	{attribute 'TcIecLibraryType'}
	{attribute 'external_name' := 'F_VN_SeparableCustomFilter_GUID_F80F76A2_7DC4_B08F_5EFC_37C20BB33E5D'}
	(* Apply a separable custom filter to the image. *)
	FUNCTION F_VN_SeparableCustomFilter : HRESULT
	VAR_INPUT
		ipSrcImage	:	ITcVnImage;	(* Source image *)
		ipDestImage	:	REFERENCE TO ITcVnImage;	(* Destination image (An appropriate destination image will be created if required.) *)
		eDestDepth	:	ETcVnElementType;	(* Destination image depth *)
	END_VAR
	VAR_IN_OUT
		stKernelX	:	TcVnMatrix;	(* 1D custom row-filter kernel with values of type REAL or LREAL *)
		stKernelY	:	TcVnMatrix;	(* 1D custom column-filter kernel with values of type REAL or LREAL *)
	END_VAR
	VAR_INPUT
		hrPrev	:	HRESULT;	(* HRESULT indicating the result of previous operations (If SUCCEEDED(hrPrev) equals false, no operation is executed.) *)
	END_VAR

END_FUNCTION

// Functions/Image Filtering/F_VN_SeparableCustomFilterExp

	{attribute 'TcIecLibraryType'}
	{attribute 'external_name' := 'F_VN_SeparableCustomFilterExp_GUID_57DB5838_7C15_B21B_75E4_43EDAA86B2A3'}
	(* Apply a separable custom filter to the image. (expert function) *)
	FUNCTION F_VN_SeparableCustomFilterExp : HRESULT
	VAR_INPUT
		ipSrcImage	:	ITcVnImage;	(* Source image *)
		ipDestImage	:	REFERENCE TO ITcVnImage;	(* Destination image (An appropriate destination image will be created if required.) *)
		eDestDepth	:	ETcVnElementType;	(* Destination image depth *)
	END_VAR
	VAR_IN_OUT
		stKernelX	:	TcVnMatrix;	(* 1D custom row-filter kernel with values of type REAL or LREAL *)
		stKernelY	:	TcVnMatrix;	(* 1D custom column-filter kernel with values of type REAL or LREAL *)
		aAnchor	:	TcVnPoint;	(* Anchor point of the kernel *)
	END_VAR
	VAR_INPUT
		fDelta	:	LREAL;	(* Value added to each pixel after filtering *)
		eBorderType	:	ETcVnBorderInterpolationMethod;	(* Image border handling *)
		hrPrev	:	HRESULT;	(* HRESULT indicating the result of previous operations (If SUCCEEDED(hrPrev) equals false, no operation is executed.) *)
	END_VAR

END_FUNCTION

// Functions/Image Filtering/F_VN_SobelFilter

	{attribute 'TcIecLibraryType'}
	{attribute 'external_name' := 'F_VN_SobelFilter_GUID_E336C8FF_820D_B834_7CC9_D468EFC4DB68'}
	(* Calculates the first, second, or mixed image derivatives using an extended Sobel filter. *)
	FUNCTION F_VN_SobelFilter : HRESULT
	VAR_INPUT
		ipSrcImage	:	ITcVnImage;	(* Source image *)
		ipDestImage	:	REFERENCE TO ITcVnImage;	(* Destination image (An appropriate destination image will be created if required.) *)
		eDestDepth	:	ETcVnElementType;	(* Destination image depth *)
		nXOrder	:	UDINT;	(* Order of the x-derivative (0, 1, 2) *)
		nYOrder	:	UDINT;	(* Order of the y-derivative (0, 1, 2) *)
		hrPrev	:	HRESULT;	(* HRESULT indicating the result of previous operations (If SUCCEEDED(hrPrev) equals false, no operation is executed.) *)
	END_VAR

END_FUNCTION

// Functions/Image Filtering/F_VN_SobelFilterExp

	{attribute 'TcIecLibraryType'}
	{attribute 'external_name' := 'F_VN_SobelFilterExp_GUID_605EE3A3_E974_B5AB_57D7_E3CF0E6E55DF'}
	(* Calculates the first, second, third, or mixed image derivatives using an extended Sobel filter. (expert function) *)
	FUNCTION F_VN_SobelFilterExp : HRESULT
	VAR_INPUT
		ipSrcImage	:	ITcVnImage;	(* Source image *)
		ipDestImage	:	REFERENCE TO ITcVnImage;	(* Destination image (An appropriate destination image will be created if required.) *)
		eDestDepth	:	ETcVnElementType;	(* Destination image depth *)
		nXOrder	:	UDINT;	(* Order of the x-derivative (must be < nKernelSize) *)
		nYOrder	:	UDINT;	(* Order of the y-derivative (must be < nKernelSize) *)
		nKernelSize	:	UDINT;	(* Size of the extended Sobel kernel (3, 5, 7, ..., 31) *)
		fScale	:	LREAL;	(* Scale factor for the computed derivative values *)
		fDelta	:	LREAL;	(* Delta value that is added to the results prior to storing them in dest *)
		eBorderType	:	ETcVnBorderInterpolationMethod;	(* Image border handling *)
		hrPrev	:	HRESULT;	(* HRESULT indicating the result of previous operations (If SUCCEEDED(hrPrev) equals false, no operation is executed.) *)
	END_VAR

END_FUNCTION

// Functions/Image Filtering/F_VN_VarianceFilter

	{attribute 'TcIecLibraryType'}
	{attribute 'external_name' := 'F_VN_VarianceFilter_GUID_E9DC81B8_162C_BF12_6F44_85E88F794313'}
	(* Calculates the local variance of an image. *)
	FUNCTION F_VN_VarianceFilter : HRESULT
	VAR_INPUT
		ipSrcImage	:	ITcVnImage;	(* Source image. Only TCVN_ET_USINT Type is supported.  *)
		ipDestImage	:	REFERENCE TO ITcVnImage;	(* Destination image of type TCVN_ET_UINT (An appropriate destination image will be created if required.) *)
		nKernelSize	:	UDINT;	(* Size of the kernel *)
		hrPrev	:	HRESULT;	(* HRESULT indicating the result of previous operations (If SUCCEEDED(hrPrev) equals false, no operation is executed.) *)
	END_VAR

END_FUNCTION

// Functions/Image Filtering/F_VN_VarianceFilterExp

	{attribute 'TcIecLibraryType'}
	{attribute 'external_name' := 'F_VN_VarianceFilterExp_GUID_A3D4813E_C46F_B737_4BEF_710F1779B2AC'}
	(* Calculates the local variance of an image. (expert function) *)
	FUNCTION F_VN_VarianceFilterExp : HRESULT
	VAR_INPUT
		ipSrcImage	:	ITcVnImage;	(* Source image. Only TCVN_ET_USINT Type is supported. *)
		ipDestImage	:	REFERENCE TO ITcVnImage;	(* Destination image of type TCVN_ET_UINT (An appropriate destination image will be created if required.) *)
		nKernelSize	:	UDINT;	(* Size of the kernel *)
		fScale	:	LREAL;	(* Scale factor for the computed variance values *)
		eBorderType	:	ETcVnBorderInterpolationMethod;	(* Image border handling *)
		hrPrev	:	HRESULT;	(* HRESULT indicating the result of previous operations (If SUCCEEDED(hrPrev) equals false, no operation is executed.) *)
	END_VAR

END_FUNCTION

// Functions/Miscellaneous/F_VN_CheckFunctionInitialization

	{attribute 'TcIecLibraryType'}
	{attribute 'external_name' := 'F_VN_CheckFunctionInitialization_GUID_C79D8AB7_DFA6_B5A0_6949_373851CC2509'}
	(* Check if a function is initialized with the specified options. *)
	FUNCTION F_VN_CheckFunctionInitialization : HRESULT
	VAR_INPUT
		eFunction	:	ETcVnInitializableFunction;	(* Initializable function *)
		nOptions	:	ULINT;	(* Initialization options for the function *)
		hrPrev	:	HRESULT;	(* HRESULT indicating the result of previous operations (If SUCCEEDED(hrPrev) equals false, no operation is executed.) *)
	END_VAR

END_FUNCTION

// Functions/Miscellaneous/F_VN_ClipLineToBoundary

	{attribute 'TcIecLibraryType'}
	{attribute 'external_name' := 'F_VN_ClipLineToBoundary_GUID_5F9D10BB_2D68_B024_7AB3_03DA1DD51379'}
	(* Clips a line to a rectangular boundary. *)
	FUNCTION F_VN_ClipLineToBoundary : HRESULT
	VAR_IN_OUT
		aLine	:	TcVnVector4_LREAL;	(* The first and second element describe the x and y component of the direction vector. The third and fourth element describe the x and y component of the position vector. *)
	END_VAR
	VAR_INPUT
		nX1	:	DINT;	(* x of top left rectangle point *)
		nY1	:	DINT;	(* y of top left rectangle point *)
		nX2	:	DINT;	(* x of bottom right rectangle point *)
		nY2	:	DINT;	(* Y of bottom right rectangle point *)
	END_VAR
	VAR_IN_OUT
		aStartPoint	:	TcVnPoint2_REAL;	(* Returns the clipped starting point of the line. *)
		aEndPoint	:	TcVnPoint2_REAL;	(* Returns the clipped end point of the line. *)
	END_VAR
	VAR_INPUT
		hrPrev	:	HRESULT;	(* HRESULT indicating the result of previous operations (If SUCCEEDED(hrPrev) equals false, no operation is executed.) *)
	END_VAR

END_FUNCTION

// Functions/Miscellaneous/F_VN_ClipLineToBoundary_ITcVnImage

	{attribute 'TcIecLibraryType'}
	{attribute 'external_name' := 'F_VN_ClipLineToBoundary_ITcVnImage_GUID_E4D5824B_2FCE_B7A7_6026_B15E63E74A8F'}
	(* Clips a line to the boundary of an image. *)
	FUNCTION F_VN_ClipLineToBoundary_ITcVnImage : HRESULT
	VAR_IN_OUT
		aLine	:	TcVnVector4_LREAL;	(* The first and second element describe the x and y component of the direction vector. The third and fourth element describe the x and y component of the position vector. *)
	END_VAR
	VAR_INPUT
		ipImage	:	ITcVnImage;	(* Image, from which to derive the boundary *)
	END_VAR
	VAR_IN_OUT
		aStartPoint	:	TcVnPoint2_REAL;	(* Returns the clipped starting point of the line. *)
		aEndPoint	:	TcVnPoint2_REAL;	(* Returns the clipped end point of the line. *)
	END_VAR
	VAR_INPUT
		hrPrev	:	HRESULT;	(* HRESULT indicating the result of previous operations (If SUCCEEDED(hrPrev) equals false, no operation is executed.) *)
	END_VAR

END_FUNCTION

// Functions/Miscellaneous/F_VN_ClipLineToBoundary_TcVnRectangle_DINT

	{attribute 'TcIecLibraryType'}
	{attribute 'external_name' := 'F_VN_ClipLineToBoundary_TcVnRectangle_DINT_GUID_87153F32_B3BD_B6D4_74D3_8036D7A03AEC'}
	(* Clips a line to a rectangular boundary. *)
	FUNCTION F_VN_ClipLineToBoundary_TcVnRectangle_DINT : HRESULT
	VAR_IN_OUT
		aLine	:	TcVnVector4_LREAL;	(* The first and second element describe the x and y component of the direction vector. The third and fourth element describe the x and y component of the position vector. *)
		stRectangle	:	TcVnRectangle_DINT;	(* Rectangular boundary *)
		aStartPoint	:	TcVnPoint2_REAL;	(* Returns the clipped starting point of the line. *)
		aEndPoint	:	TcVnPoint2_REAL;	(* Returns the clipped end point of the line. *)
	END_VAR
	VAR_INPUT
		hrPrev	:	HRESULT;	(* HRESULT indicating the result of previous operations (If SUCCEEDED(hrPrev) equals false, no operation is executed.) *)
	END_VAR

END_FUNCTION

// Functions/Miscellaneous/F_VN_ConvertITcUnknownToITcVnBitmapExport

	{attribute 'TcIecLibraryType'}
	{attribute 'external_name' := 'F_VN_ConvertITcUnknownToITcVnBitmapExport_GUID_2EB3F845_B1C8_B651_6556_4CA6475660E3'}
	(* Convert an ITcUnknown interface pointer to an ITcVnBitmapExport interface pointer. The destination pointer will be released (if existing) and set to the source pointer. The source pointer will be set to 0. *)
	FUNCTION F_VN_ConvertITcUnknownToITcVnBitmapExport : HRESULT
	VAR_INPUT
		ipSrc	:	REFERENCE TO ITcUnknown;	(* Source pointer *)
		ipDest	:	REFERENCE TO ITcVnBitmapExport;	(* Destination pointer *)
		hrPrev	:	HRESULT;	(* HRESULT indicating the result of previous operations (If SUCCEEDED(hrPrev) equals false, no operation is executed.) *)
	END_VAR

END_FUNCTION

// Functions/Miscellaneous/F_VN_ConvertITcUnknownToITcVnContainer

	{attribute 'TcIecLibraryType'}
	{attribute 'external_name' := 'F_VN_ConvertITcUnknownToITcVnContainer_GUID_138FA1B4_D6BC_B0DA_5E49_0E92D1E26E82'}
	(* Convert an ITcUnknown interface pointer to an ITcVnContainer interface pointer. The destination pointer will be released (if existing) and set to the source pointer. The source pointer will be set to 0. *)
	FUNCTION F_VN_ConvertITcUnknownToITcVnContainer : HRESULT
	VAR_INPUT
		ipSrc	:	REFERENCE TO ITcUnknown;	(* Source pointer *)
		ipDest	:	REFERENCE TO ITcVnContainer;	(* Destination pointer *)
		hrPrev	:	HRESULT;	(* HRESULT indicating the result of previous operations (If SUCCEEDED(hrPrev) equals false, no operation is executed.) *)
	END_VAR

END_FUNCTION

// Functions/Miscellaneous/F_VN_ConvertITcUnknownToITcVnImage

	{attribute 'TcIecLibraryType'}
	{attribute 'external_name' := 'F_VN_ConvertITcUnknownToITcVnImage_GUID_1C77EE9B_F836_B880_71E3_3B6B684F7DE7'}
	(* Convert an ITcUnknown interface pointer to an ITcVnImage interface pointer. The destination pointer will be released (if existing) and set to the source pointer. The source pointer will be set to 0. *)
	FUNCTION F_VN_ConvertITcUnknownToITcVnImage : HRESULT
	VAR_INPUT
		ipSrc	:	REFERENCE TO ITcUnknown;	(* Source pointer *)
		ipDest	:	REFERENCE TO ITcVnImage;	(* Destination pointer *)
		hrPrev	:	HRESULT;	(* HRESULT indicating the result of previous operations (If SUCCEEDED(hrPrev) equals false, no operation is executed.) *)
	END_VAR

END_FUNCTION

// Functions/Miscellaneous/F_VN_ConvertITcUnknownToITcVnMlModel

	{attribute 'TcIecLibraryType'}
	{attribute 'external_name' := 'F_VN_ConvertITcUnknownToITcVnMlModel_GUID_00F937E1_B5BF_BE31_604E_B90F05C045F2'}
	(* Convert an ITcUnknown interface pointer to an ITcVnMlModel interface pointer. The destination pointer will be released (if existing) and set to the source pointer. The source pointer will be set to 0. *)
	FUNCTION F_VN_ConvertITcUnknownToITcVnMlModel : HRESULT
	VAR_INPUT
		ipSrc	:	REFERENCE TO ITcUnknown;	(* Source pointer *)
		ipDest	:	REFERENCE TO ITcVnMlModel;	(* Destination pointer *)
		hrPrev	:	HRESULT;	(* HRESULT indicating the result of previous operations (If SUCCEEDED(hrPrev) equals false, no operation is executed.) *)
	END_VAR

END_FUNCTION

// Functions/Miscellaneous/F_VN_DeinitializeFunction

	{attribute 'TcIecLibraryType'}
	{attribute 'external_name' := 'F_VN_DeinitializeFunction_GUID_3AEC9F0B_9689_B047_59F3_4962202BFD13'}
	(* Deinitialize the specified options for the function. *)
	FUNCTION F_VN_DeinitializeFunction : HRESULT
	VAR_INPUT
		eFunction	:	ETcVnInitializableFunction;	(* Initializable function *)
		nOptions	:	ULINT;	(* Initialization options for the function *)
		hrPrev	:	HRESULT;	(* HRESULT indicating the result of previous operations (If SUCCEEDED(hrPrev) equals false, no operation is executed.) *)
	END_VAR

END_FUNCTION

// Functions/Miscellaneous/F_VN_GetTimestamp

	{attribute 'TcIecLibraryType'}
	{attribute 'external_name' := 'F_VN_GetTimestamp_GUID_C6774F0F_1FD8_B43F_4215_84A6E64C27D7'}
	(* Get the timestamp (actual DC time) from the last change of an object (e.g. ITcVnImage or ITcVnContainer) *)
	FUNCTION F_VN_GetTimestamp : HRESULT
	VAR_INPUT
		ipUnknown	:	ITcUnknown;	(* An object implementing ITcUnknown and ITcVnTimestamp (e.g. ITcVnImage or ITcVnContainer) *)
	END_VAR
	VAR_IN_OUT
		nTimestamp	:	LINT;	(* Returns the timestamp *)
	END_VAR
	VAR_INPUT
		hrPrev	:	HRESULT;	(* HRESULT indicating the result of previous operations (If SUCCEEDED(hrPrev) equals false, no operation is executed.) *)
	END_VAR

END_FUNCTION

// Functions/Miscellaneous/F_VN_HuMomentInvariants

	{attribute 'TcIecLibraryType'}
	{attribute 'external_name' := 'F_VN_HuMomentInvariants_GUID_BC907807_859C_B8CF_4281_4253B572D82F'}
	(* Computes the Hu moment invariants. *)
	FUNCTION F_VN_HuMomentInvariants : HRESULT
	VAR_IN_OUT
		stMoments	:	TcVnMoments;	(* Moments from which to compute the Hu invariants *)
		aHuInvariants	:	TcVnArray7_LREAL;	(* Returns the Hu moment invariants *)
	END_VAR
	VAR_INPUT
		hrPrev	:	HRESULT;	(* HRESULT indicating the result of previous operations (If SUCCEEDED(hrPrev) equals false, no operation is executed.) *)
	END_VAR

END_FUNCTION

// Functions/Miscellaneous/F_VN_InitMatrixStruct

	{attribute 'TcIecLibraryType'}
	{attribute 'external_name' := 'F_VN_InitMatrixStruct_GUID_8788B85B_B119_B982_4540_76E6A59BE885'}
	(* Initialize a struct of the type TcVnMatrix extending a buffer with metainformation so that it can be used as a matrix. *)
	FUNCTION F_VN_InitMatrixStruct : HRESULT
	VAR_INPUT
		pSrcBuffer	:	PVOID;	(* Source buffer *)
	END_VAR
	VAR_IN_OUT
		stDestMatrix	:	TcVnMatrix;	(* Returns completed matrix struct *)
	END_VAR
	VAR_INPUT
		nRows	:	UDINT;	(* Matrix rows *)
		nCols	:	UDINT;	(* Matrix columns *)
		eElementType	:	ETcVnElementType;	(* Type of the matrix elements *)
		hrPrev	:	HRESULT;	(* HRESULT indicating the result of previous operations (If SUCCEEDED(hrPrev) equals false, no operation is executed.) *)
	END_VAR

END_FUNCTION

// Functions/Miscellaneous/F_VN_InvertMatrix3x3

	{attribute 'TcIecLibraryType'}
	{attribute 'external_name' := 'F_VN_InvertMatrix3x3_GUID_E8B1B6D0_88FB_BEBB_7DCF_DBFDBEA44864'}
	(* Invert a 3x3 matrix. *)
	FUNCTION F_VN_InvertMatrix3x3 : HRESULT
	VAR_IN_OUT
		aSrcMatrix	:	TcVnMatrix3x3_LREAL;	(* Source matrix *)
		aInvertedMatrix	:	TcVnMatrix3x3_LREAL;	(* Returns inverted matrix *)
	END_VAR
	VAR_INPUT
		hrPrev	:	HRESULT;	(* HRESULT indicating the result of previous operations (If SUCCEEDED(hrPrev) equals false, no operation is executed.) *)
	END_VAR

END_FUNCTION

// Functions/Miscellaneous/F_VN_LineIntersectionPoint

	{attribute 'TcIecLibraryType'}
	{attribute 'external_name' := 'F_VN_LineIntersectionPoint_GUID_09DE1F0A_AD0F_BD48_4A68_F123E5CFE511'}
	(* Computes the intersection point between two lines (returns S_FALSE if the provided lines are parallel). *)
	FUNCTION F_VN_LineIntersectionPoint : HRESULT
	VAR_IN_OUT
		aLine1	:	TcVnVector4_LREAL;	(* First line. The first and second element describe the x and y component of a vector collinear to the line. The third and fourth element describe the x and y component of a point on the line. *)
		aLine2	:	TcVnVector4_LREAL;	(* Second line. The first and second element describe the x and y component of a vector collinear to the line. The third and fourth element describe the x and y component of a point on the line. *)
		aIntersecPoint	:	TcVnPoint2_REAL;	(* Returns the intersection point of aLine1 and aLine2. *)
	END_VAR
	VAR_INPUT
		hrPrev	:	HRESULT;	(* HRESULT indicating the result of previous operations (If SUCCEEDED(hrPrev) equals false, no operation is executed.) *)
	END_VAR

END_FUNCTION

// Functions/Miscellaneous/F_VN_LineIntersectionPointAndAngle

	{attribute 'TcIecLibraryType'}
	{attribute 'external_name' := 'F_VN_LineIntersectionPointAndAngle_GUID_02ACE12C_D7B0_BC9D_4D49_0FA5929B3128'}
	(* Computes the intersection point and angle between two lines (returns S_FALSE if the provided lines are parallel). *)
	FUNCTION F_VN_LineIntersectionPointAndAngle : HRESULT
	VAR_IN_OUT
		aLine1	:	TcVnVector4_LREAL;	(* First line. The first and second element describe the x and y component of a vector collinear to the line. The third and fourth element describe the x and y component of a point on the line. *)
		aLine2	:	TcVnVector4_LREAL;	(* Second line. The first and second element describe the x and y component of a vector collinear to the line. The third and fourth element describe the x and y component of a point on the line. *)
		aIntersecPoint	:	TcVnPoint2_REAL;	(* Returns the intersection point of aLine1 and aLine2. *)
		fAngle	:	REAL;	(* Returns the intersection angle of aLine1 and aLine2. *)
	END_VAR
	VAR_INPUT
		bAngleInDegrees	:	BOOL;	(* If TRUE, fAngle is in degrees. If FALSE, fAngle is in radians. *)
		hrPrev	:	HRESULT;	(* HRESULT indicating the result of previous operations (If SUCCEEDED(hrPrev) equals false, no operation is executed.) *)
	END_VAR

END_FUNCTION

// Functions/Miscellaneous/F_VN_MultiplyMatrices

	{attribute 'TcIecLibraryType'}
	{attribute 'external_name' := 'F_VN_MultiplyMatrices_GUID_EE5BE0D3_B880_BE84_491F_D1628BE189AD'}
	(* Matrix multiplication of two matrices (A * B = C). All matrices are represented by structs holding a pointer to an array of the appropriate size. *)
	FUNCTION F_VN_MultiplyMatrices : HRESULT
	VAR_IN_OUT
		stSrcMatrix1	:	TcVnMatrix;	(* First source matrix (A) *)
		stSrcMatrix2	:	TcVnMatrix;	(* Second source matrix (B) *)
		stDestMatrix	:	TcVnMatrix;	(* Destination matrix (C) (The destination matrix is filled by this function, but the required memory needs to be provided.) *)
	END_VAR
	VAR_INPUT
		hrPrev	:	HRESULT;	(* HRESULT indicating the result of previous operations (If SUCCEEDED(hrPrev) equals false, no operation is executed.) *)
	END_VAR

END_FUNCTION

// Functions/Miscellaneous/F_VN_RotatedRectangleCorners

	{attribute 'TcIecLibraryType'}
	{attribute 'external_name' := 'F_VN_RotatedRectangleCorners_GUID_3231DEDE_31EB_BE6F_5229_2987A4B74C79'}
	(* Computes the 4 corner points of a rotated rectangle. *)
	FUNCTION F_VN_RotatedRectangleCorners : HRESULT
	VAR_IN_OUT
		stRect	:	TcVnRotatedRectangle;	(* Rotated rectangle *)
		aCorners	:	TcVnArray4_Point2_REAL;	(* Returns the 4 corner points *)
	END_VAR
	VAR_INPUT
		hrPrev	:	HRESULT;	(* HRESULT indicating the result of previous operations (If SUCCEEDED(hrPrev) equals false, no operation is executed.) *)
	END_VAR

END_FUNCTION

// Functions/Miscellaneous/F_VN_RotatedRectangleIntersection

	{attribute 'TcIecLibraryType'}
	{attribute 'external_name' := 'F_VN_RotatedRectangleIntersection_GUID_9F7F4134_1F97_B2F4_54BC_78B2002BD86F'}
	(* Finds the intersection of 2 rotated rectangles. *)
	FUNCTION F_VN_RotatedRectangleIntersection : HRESULT
	VAR_IN_OUT
		stRect1	:	TcVnRotatedRectangle;	(* Rotated rectangle 1 *)
		stRect2	:	TcVnRotatedRectangle;	(* Rotated rectangle 2 *)
	END_VAR
	VAR_INPUT
		ipIntersection	:	REFERENCE TO ITcVnContainer;	(* Returns the intersection points (ContainerType_Vector_TcVnPoint2_REAL, non-zero interface pointers are reused) *)
	END_VAR
	VAR_IN_OUT
		eIntersection	:	ETcVnRectangleIntersection;	(* Returns the intersection type *)
	END_VAR
	VAR_INPUT
		hrPrev	:	HRESULT;	(* HRESULT indicating the result of previous operations (If SUCCEEDED(hrPrev) equals false, no operation is executed.) *)
	END_VAR

END_FUNCTION

// Functions/Miscellaneous/F_VN_SetRngSeed

	{attribute 'TcIecLibraryType'}
	{attribute 'external_name' := 'F_VN_SetRngSeed_GUID_898DFC81_C65B_B1C7_5C81_FA6D845A134F'}
	(* Sets the internal pseudo random number generator seed (intended for testing purposes only). *)
	FUNCTION F_VN_SetRngSeed : HRESULT
	VAR_INPUT
		nSeed	:	DINT;	(* seed (0 sets the generator back to its initial state) *)
		hrPrev	:	HRESULT;	(* HRESULT indicating the result of previous operations (If SUCCEEDED(hrPrev) equals false, no operation is executed.) *)
	END_VAR

END_FUNCTION

// Functions/Miscellaneous/F_VN_UpdateTimestamp

	{attribute 'TcIecLibraryType'}
	{attribute 'external_name' := 'F_VN_UpdateTimestamp_GUID_5FA1F89A_14B5_BE95_6D78_BFBBBB9A3BDA'}
	(* Update the timestamp of an object to the actual DC time (e.g. ITcVnImage or ITcVnContainer) *)
	FUNCTION F_VN_UpdateTimestamp : HRESULT
	VAR_INPUT
		ipUnknown	:	ITcUnknown;	(* An object implementing ITcUnknown and ITcVnTimestamp (e.g. ITcVnImage or ITcVnContainer) *)
		hrPrev	:	HRESULT;	(* HRESULT indicating the result of previous operations (If SUCCEEDED(hrPrev) equals false, no operation is executed.) *)
	END_VAR

END_FUNCTION

// Functions/Basic Image Operations/F_VN_CombineImageChannels

	{attribute 'TcIecLibraryType'}
	{attribute 'external_name' := 'F_VN_CombineImageChannels_GUID_CEC59215_B089_B2AA_5669_42D9A49D5EE8'}
	(* Combines several single-channel images into one multi-channel image. *)
	FUNCTION F_VN_CombineImageChannels : HRESULT
	VAR_INPUT
		pSrcImages	:	PVOID;	(* Pointer to an array of single-channel source images *)
		ipDestImage	:	REFERENCE TO ITcVnImage;	(* Multi-channel destination image (An appropriate destination image will be created if required.) *)
		nSrcArraySize	:	UINT;	(* pSrcImages array size *)
		hrPrev	:	HRESULT;	(* HRESULT indicating the result of previous operations (If SUCCEEDED(hrPrev) equals false, no operation is executed.) *)
	END_VAR

END_FUNCTION

// Functions/Basic Image Operations/F_VN_ConvertElementType

	{attribute 'TcIecLibraryType'}
	{attribute 'external_name' := 'F_VN_ConvertElementType_GUID_6F7F69F6_5FC0_BB1A_7DD0_18A20D6CEE8C'}
	(* Converts an image to another element type. *)
	FUNCTION F_VN_ConvertElementType : HRESULT
	VAR_INPUT
		ipSrcImage	:	ITcVnImage;	(* Source image *)
		ipDestImage	:	REFERENCE TO ITcVnImage;	(* Destination image (An appropriate destination image will be created if required.) *)
		eElementType	:	ETcVnElementType;	(* Desired element type of the destination image *)
		hrPrev	:	HRESULT;	(* HRESULT indicating the result of previous operations (If SUCCEEDED(hrPrev) equals false, no operation is executed.) *)
	END_VAR

END_FUNCTION

// Functions/Basic Image Operations/F_VN_ConvertElementTypeExp

	{attribute 'TcIecLibraryType'}
	{attribute 'external_name' := 'F_VN_ConvertElementTypeExp_GUID_9F88F6DC_3EAC_B7E7_64C9_02A04E70F2D7'}
	(* Converts an image to another element type. (expert function) *)
	FUNCTION F_VN_ConvertElementTypeExp : HRESULT
	VAR_INPUT
		ipSrcImage	:	ITcVnImage;	(* Source image *)
		ipDestImage	:	REFERENCE TO ITcVnImage;	(* Destination image (An appropriate destination image will be created if required.) *)
		eElementType	:	ETcVnElementType;	(* Desired element type of the destination image *)
		fScaleFactor	:	LREAL;	(* Scale factor for the pixel values *)
		fDelta	:	LREAL;	(* Value that is added to the scaled pixel values *)
		hrPrev	:	HRESULT;	(* HRESULT indicating the result of previous operations (If SUCCEEDED(hrPrev) equals false, no operation is executed.) *)
	END_VAR

END_FUNCTION

// Functions/Basic Image Operations/F_VN_CopyImage

	{attribute 'TcIecLibraryType'}
	{attribute 'external_name' := 'F_VN_CopyImage_GUID_31D085A7_0879_B268_4E18_6515F2A9E514'}
	(* Creates a deep copy of an image. *)
	FUNCTION F_VN_CopyImage : HRESULT
	VAR_INPUT
		ipSrcImage	:	ITcVnImage;	(* Source image *)
		ipDestImage	:	REFERENCE TO ITcVnImage;	(* Destination image (An appropriate destination image will be created if required.) *)
		hrPrev	:	HRESULT;	(* HRESULT indicating the result of previous operations (If SUCCEEDED(hrPrev) equals false, no operation is executed.) *)
	END_VAR

END_FUNCTION

// Functions/Basic Image Operations/F_VN_CopyImageRegion

	{attribute 'TcIecLibraryType'}
	{attribute 'external_name' := 'F_VN_CopyImageRegion_GUID_08E0E4FC_176C_B0B4_7DD0_8290BD7750BB'}
	(* Deep copy the specified region of interest into a new image. *)
	FUNCTION F_VN_CopyImageRegion : HRESULT
	VAR_INPUT
		ipSrcImage	:	ITcVnImage;	(* Source image *)
		nX	:	UDINT;	(* Left boundary (inclusive 0-based index) *)
		nY	:	UDINT;	(* Upper boundary (inclusive 0-based index) *)
		nWidth	:	UDINT;	(* ROI width *)
		nHeight	:	UDINT;	(* ROI height *)
		ipDestImage	:	REFERENCE TO ITcVnImage;	(* Destination image (An appropriate destination image will be created if required.) *)
		hrPrev	:	HRESULT;	(* HRESULT indicating the result of previous operations (If SUCCEEDED(hrPrev) equals false, no operation is executed.) *)
	END_VAR

END_FUNCTION

// Functions/Basic Image Operations/F_VN_CopyImageRegionToRegion

	{attribute 'TcIecLibraryType'}
	{attribute 'external_name' := 'F_VN_CopyImageRegionToRegion_GUID_9FCFE978_4BC7_B205_57F3_9126424D30C1'}
	(* Copy an image region into another image region. *)
	FUNCTION F_VN_CopyImageRegionToRegion : HRESULT
	VAR_INPUT
		ipSrcImage	:	ITcVnImage;	(* Source image *)
		nXSrc	:	UDINT;	(* Left boundary in ipSrcImage (inclusive 0-based index) *)
		nYSrc	:	UDINT;	(* Upper boundary in ipSrcImage (inclusive 0-based index) *)
		nWidth	:	UDINT;	(* ROI width *)
		nHeight	:	UDINT;	(* ROI height *)
		ipDestImage	:	ITcVnImage;	(* Destination image (same type as ipSrcImage) *)
		nXDest	:	UDINT;	(* Left boundary in ipDestImage (inclusive 0-based index) *)
		nYDest	:	UDINT;	(* Upper boundary in ipDestImage (inclusive 0-based index) *)
		hrPrev	:	HRESULT;	(* HRESULT indicating the result of previous operations (If SUCCEEDED(hrPrev) equals false, no operation is executed.) *)
	END_VAR

END_FUNCTION

// Functions/Basic Image Operations/F_VN_CopyIntoDisplayableImage

	{attribute 'TcIecLibraryType'}
	{attribute 'external_name' := 'F_VN_CopyIntoDisplayableImage_GUID_9B5ACD8B_7A74_B136_4B36_29B5402D29AD'}
	(* Copys an image into a displayable image. If you do not want to use ipSrcImage after this function call, you might want to use F_VN_TransformIntoDisplayableImage instead for better performance. *)
	FUNCTION F_VN_CopyIntoDisplayableImage : HRESULT
	VAR_INPUT
		ipSrcImage	:	ITcVnImage;	(* Source image *)
		ipDestImage	:	REFERENCE TO ITcVnDisplayableImage;	(* Returns the displayable image *)
		hrPrev	:	HRESULT;	(* HRESULT indicating the result of previous operations (If SUCCEEDED(hrPrev) equals false, no operation is executed.) *)
	END_VAR

END_FUNCTION

// Functions/Basic Image Operations/F_VN_TransformIntoDisplayableImage

	{attribute 'TcIecLibraryType'}
	{attribute 'external_name' := 'F_VN_TransformIntoDisplayableImage_GUID_6AD45584_205E_B216_5C58_56CBDB012F18'}
	(* Transform an image into a displayable image. The source image will be released and zeroed while existing destination images will be released and overwritten with the function result. The source image must not be used anywhere else and the transformation is very fast. If you want to use ipSrcImage after this function call, use F_VN_CopyIntoDisplayableImage instead. *)
	FUNCTION F_VN_TransformIntoDisplayableImage : HRESULT
	VAR_INPUT
		ipSrcImage	:	REFERENCE TO ITcVnImage;	(* Source image *)
		ipDestImage	:	REFERENCE TO ITcVnDisplayableImage;	(* Returns the displayable image *)
		hrPrev	:	HRESULT;	(* HRESULT indicating the result of previous operations (If SUCCEEDED(hrPrev) equals false, no operation is executed.) *)
	END_VAR

END_FUNCTION

// Functions/Basic Image Operations/F_VN_CreateAssociatedImage

	{attribute 'TcIecLibraryType'}
	{attribute 'external_name' := 'F_VN_CreateAssociatedImage_GUID_28E7076C_C03E_B354_6911_32162133E233'}
	(* Creates a new image that shares its data with the source image. E.g. useful to work on different (disjoint) ROIs in parallel. *)
	FUNCTION F_VN_CreateAssociatedImage : HRESULT
	VAR_INPUT
		ipSrcImage	:	ITcVnImage;	(* Source image *)
		ipDestImage	:	REFERENCE TO ITcVnImage;	(* Returns the created image (Non-zero interface pointers are reused.) *)
		hrPrev	:	HRESULT;	(* HRESULT indicating the result of previous operations (If SUCCEEDED(hrPrev) equals false, no operation is executed.) *)
	END_VAR

END_FUNCTION

// Functions/Basic Image Operations/F_VN_CreateEmptyImage

	{attribute 'TcIecLibraryType'}
	{attribute 'external_name' := 'F_VN_CreateEmptyImage_GUID_EFEA92DB_41B7_B325_5636_D57075778D40'}
	(* Creates an empty image without allocating any data buffer. The initial reference count is set to one if a new image interface is created and kept, otherwise. *)
	FUNCTION F_VN_CreateEmptyImage : HRESULT
	VAR_INPUT
		ipImage	:	REFERENCE TO ITcVnImage;	(* Returns the created image *)
		hrPrev	:	HRESULT;	(* HRESULT indicating the result of previous operations (If SUCCEEDED(hrPrev) equals false, no operation is executed.) *)
	END_VAR

END_FUNCTION

// Functions/Basic Image Operations/F_VN_CreateImage

	{attribute 'TcIecLibraryType'}
	{attribute 'external_name' := 'F_VN_CreateImage_GUID_E5409511_83E7_BBC5_6049_5D6C960F853B'}
	(* Creates an image and allocate an appropriate data buffer. The initial reference count is set to one if a new image interface is created and kept, otherwise. *)
	FUNCTION F_VN_CreateImage : HRESULT
	VAR_INPUT
		ipImage	:	REFERENCE TO ITcVnImage;	(* Returns the created image (Non-zero interface pointers are reused.) *)
		nWidth	:	UDINT;	(* Image width *)
		nHeight	:	UDINT;	(* Image height *)
		ePixelType	:	ETcVnElementType;	(* Pixel type *)
		nChannelNum	:	UDINT;	(* Number of channels (1 to 255) *)
		hrPrev	:	HRESULT;	(* HRESULT indicating the result of previous operations (If SUCCEEDED(hrPrev) equals false, no operation is executed.) *)
	END_VAR

END_FUNCTION

// Functions/Basic Image Operations/F_VN_CreateImageAndSetPixels

	{attribute 'TcIecLibraryType'}
	{attribute 'external_name' := 'F_VN_CreateImageAndSetPixels_GUID_C0A6BA34_6341_B2CA_61DB_1D04E2B200F2'}
	(* Creates an image, allocates an appropriate data buffer and sets all pixels to the specified value. The initial reference count is set to one if a new image interface is created and kept, otherwise. *)
	FUNCTION F_VN_CreateImageAndSetPixels : HRESULT
	VAR_INPUT
		ipImage	:	REFERENCE TO ITcVnImage;	(* Returns the created image (Non-zero interface pointers are reused.) *)
		nWidth	:	UDINT;	(* Image width *)
		nHeight	:	UDINT;	(* Image height *)
		ePixelType	:	ETcVnElementType;	(* Pixel type *)
		nChannelNum	:	UDINT;	(* Number of channels (1 to 4) *)
	END_VAR
	VAR_IN_OUT
		aValue	:	TcVnVector4_LREAL;	(* Pixel value *)
	END_VAR
	VAR_INPUT
		hrPrev	:	HRESULT;	(* HRESULT indicating the result of previous operations (If SUCCEEDED(hrPrev) equals false, no operation is executed.) *)
	END_VAR

END_FUNCTION

// Functions/Basic Image Operations/F_VN_CreateImageFromArray

	{attribute 'TcIecLibraryType'}
	{attribute 'external_name' := 'F_VN_CreateImageFromArray_GUID_09F968F2_FDD1_BEA0_607E_911658E8A95D'}
	(* Creates an image and initialize it with the provided data. The initial reference count is set to one if a new image interface is created and kept, otherwise. *)
	FUNCTION F_VN_CreateImageFromArray : HRESULT
	VAR_INPUT
		pData	:	PVOID;	(* Pointer to the 1D data array. Make sure that the array contains at least nWidth * nHeight * nChannelNum elements and that the array element type matches ePixelType. *)
		ipImage	:	REFERENCE TO ITcVnImage;	(* Returns the created image (Non-zero interface pointers are reused.) *)
		nWidth	:	UDINT;	(* Image width *)
		nHeight	:	UDINT;	(* Image height *)
		ePixelType	:	ETcVnElementType;	(* Pixel type *)
		nChannelNum	:	UDINT;	(* Number of channels (1 to 255) *)
		hrPrev	:	HRESULT;	(* HRESULT indicating the result of previous operations (If SUCCEEDED(hrPrev) equals false, no operation is executed.) *)
	END_VAR

END_FUNCTION

// Functions/Basic Image Operations/F_VN_ExportImage

	{attribute 'TcIecLibraryType'}
	{attribute 'external_name' := 'F_VN_ExportImage_GUID_7AA7CB67_E83B_B7C2_6BF1_DAD6E2F3360E'}
	(* Exports the image data into a given buffer (e.g. an array). F_VN_ExportImageSize should be called before to get the required buffer size. *)
	FUNCTION F_VN_ExportImage : HRESULT
	VAR_INPUT
		ipImage	:	ITcVnImage;	(* Image *)
		pBuffer	:	PVOID;	(* Pointer to a buffer to store the image data (Make sure to allocate enough memory! The required size in bytes can be determined using the function F_VN_ExportImageSize) *)
		nBufferSize	:	ULINT;	(* Size of the buffer memory in bytes *)
		hrPrev	:	HRESULT;	(* HRESULT indicating the result of previous operations (If SUCCEEDED(hrPrev) equals false, no operation is executed.) *)
	END_VAR

END_FUNCTION

// Functions/Basic Image Operations/F_VN_ExportImageSize

	{attribute 'TcIecLibraryType'}
	{attribute 'external_name' := 'F_VN_ExportImageSize_GUID_F118B591_1AEC_B881_4C93_1CB889CF694D'}
	(* Get the required buffer size (in bytes) to store the image data. *)
	FUNCTION F_VN_ExportImageSize : HRESULT
	VAR_INPUT
		ipImage	:	ITcVnImage;	(* Image *)
	END_VAR
	VAR_IN_OUT
		nBufferSize	:	ULINT;	(* Returns the required buffer size in bytes *)
	END_VAR
	VAR_INPUT
		hrPrev	:	HRESULT;	(* HRESULT indicating the result of previous operations (If SUCCEEDED(hrPrev) equals false, no operation is executed.) *)
	END_VAR

END_FUNCTION

// Functions/Basic Image Operations/F_VN_ExportImageAsBmp

	{attribute 'TcIecLibraryType'}
	{attribute 'external_name' := 'F_VN_ExportImageAsBmp_GUID_23FE3C48_3CAF_B978_4536_643BF65CA576'}
	(* Exports the image as bitmap into a given buffer (e.g. an array). F_VN_ExportImageAsBmpSize should be called before to get the required buffer size. *)
	FUNCTION F_VN_ExportImageAsBmp : HRESULT
	VAR_INPUT
		ipImage	:	ITcVnImage;	(* Image *)
		pBuffer	:	PVOID;	(* Pointer to a buffer to store the bitmap image (Make sure to allocate enough memory! The required size in bytes can be determined using the function F_VN_ExportImageAsBmpSize) *)
		nBufferSize	:	ULINT;	(* Size of the buffer memory in bytes *)
		hrPrev	:	HRESULT;	(* HRESULT indicating the result of previous operations (If SUCCEEDED(hrPrev) equals false, no operation is executed.) *)
	END_VAR

END_FUNCTION

// Functions/Basic Image Operations/F_VN_ExportImageAsBmpSize

	{attribute 'TcIecLibraryType'}
	{attribute 'external_name' := 'F_VN_ExportImageAsBmpSize_GUID_67ED4571_3245_B415_5F0F_DF2DB73B983A'}
	(* Get the required buffer size (in bytes) to store the image as bitmap. *)
	FUNCTION F_VN_ExportImageAsBmpSize : HRESULT
	VAR_INPUT
		ipImage	:	ITcVnImage;	(* Image *)
	END_VAR
	VAR_IN_OUT
		nBufferSize	:	ULINT;	(* Returns the required buffer size in bytes *)
	END_VAR
	VAR_INPUT
		hrPrev	:	HRESULT;	(* HRESULT indicating the result of previous operations (If SUCCEEDED(hrPrev) equals false, no operation is executed.) *)
	END_VAR

END_FUNCTION

// Functions/Basic Image Operations/F_VN_ExportImageAsBmpExp

	{attribute 'TcIecLibraryType'}
	{attribute 'external_name' := 'F_VN_ExportImageAsBmpExp_GUID_2F47A87A_3F9B_B025_76EC_078003AF02E0'}
	(* Exports the image as bitmap into a given buffer (e.g. an array). F_VN_ExportImageAsBmpSizeExp should be called before to get the required buffer size. (expert function) *)
	FUNCTION F_VN_ExportImageAsBmpExp : HRESULT
	VAR_INPUT
		ipImage	:	ITcVnImage;	(* Image *)
		pBuffer	:	PVOID;	(* Pointer to a buffer to store the bitmap image (Make sure to allocate enough memory! The required size in bytes can be determined using the function F_VN_ExportImageAsBmpSizeExp) *)
		nBufferSize	:	ULINT;	(* Size of the buffer memory in bytes *)
		nWidth	:	UDINT;	(* Desired width (or 0 to keep the original width) *)
		nHeight	:	UDINT;	(* Desired height (or 0 to keep the original height) *)
		hrPrev	:	HRESULT;	(* HRESULT indicating the result of previous operations (If SUCCEEDED(hrPrev) equals false, no operation is executed.) *)
	END_VAR

END_FUNCTION

// Functions/Basic Image Operations/F_VN_ExportImageAsBmpSizeExp

	{attribute 'TcIecLibraryType'}
	{attribute 'external_name' := 'F_VN_ExportImageAsBmpSizeExp_GUID_7D1E35BF_FC52_B2B0_4AF6_04E042DC3A1E'}
	(* Get the required buffer size (in bytes) to store the image as bitmap. (expert function) *)
	FUNCTION F_VN_ExportImageAsBmpSizeExp : HRESULT
	VAR_INPUT
		ipImage	:	ITcVnImage;	(* Image *)
	END_VAR
	VAR_IN_OUT
		nBufferSize	:	ULINT;	(* Returns the required buffer size in bytes *)
	END_VAR
	VAR_INPUT
		nWidth	:	UDINT;	(* Desired width (or 0 to keep the original width) *)
		nHeight	:	UDINT;	(* Desired height (or 0 to keep the original height) *)
		hrPrev	:	HRESULT;	(* HRESULT indicating the result of previous operations (If SUCCEEDED(hrPrev) equals false, no operation is executed.) *)
	END_VAR

END_FUNCTION

// Functions/Basic Image Operations/F_VN_FuseImages

	{attribute 'TcIecLibraryType'}
	{attribute 'external_name' := 'F_VN_FuseImages_GUID_2CC3835F_7164_B79D_5473_4B08516F7B7C'}
	(* Fuse 2 images vertically (intended for line scan cameras). *)
	FUNCTION F_VN_FuseImages : HRESULT
	VAR_INPUT
		ipSrcImage1	:	ITcVnImage;	(* Source image 1 *)
		ipSrcImage2	:	ITcVnImage;	(* Source image 2 *)
		ipDestImage	:	REFERENCE TO ITcVnImage;	(* Destination image *)
		nFirstLine	:	UDINT;	(* Line index in ipSrcImage1, which is the first line in ipDestImage *)
		nNumLines	:	UDINT;	(* The number of lines that should be copied to ipDestImage, starting with nFirstLine in ipSrcImage1. Once the last line of ipSrcImage1 was copied, the remaining lines are copied from ipSrcImage2, starting at line index 0. *)
		hrPrev	:	HRESULT;	(* HRESULT indicating the result of previous operations (If SUCCEEDED(hrPrev) equals false, no operation is executed.) *)
	END_VAR

END_FUNCTION

// Functions/Basic Image Operations/F_VN_FuseImagesArray

	{attribute 'TcIecLibraryType'}
	{attribute 'external_name' := 'F_VN_FuseImagesArray_GUID_18CAE4B4_69F5_B090_5098_443C680EAE36'}
	(* Fuse up to 10 images vertically (intended for line scan cameras). *)
	FUNCTION F_VN_FuseImagesArray : HRESULT
	VAR_IN_OUT
		aSrcImageArray	:	TcVnArray10_ITcVnImage;	(* Ten-element source image array (not all elements need to be filled, nValidImages specifies the actual amount of images) *)
	END_VAR
	VAR_INPUT
		nValidImages	:	UDINT;	(* Number of valid images in aSrcImageArray *)
		ipDestImage	:	REFERENCE TO ITcVnImage;	(* Destination image *)
		nFirstLine	:	UDINT;	(* Line index in ipSrcImage1, which is the first line in ipDestImage *)
		nNumLines	:	UDINT;	(* The number of lines that should be copied to ipDestImage, starting with nFirstLine in aSrcImageArray[0]. Once the last line of aSrcImageArray[0] was copied, the remaining lines are copied from aSrcImageArray[1] (starting at line index 0) and so on. *)
		hrPrev	:	HRESULT;	(* HRESULT indicating the result of previous operations (If SUCCEEDED(hrPrev) equals false, no operation is executed.) *)
	END_VAR

END_FUNCTION

// Functions/Basic Image Operations/F_VN_GetImageChannel

	{attribute 'TcIecLibraryType'}
	{attribute 'external_name' := 'F_VN_GetImageChannel_GUID_7D2D9648_51FE_B416_6D0F_FE2AC8E616C5'}
	(* Return the specified source image channel as a single-channel image. *)
	FUNCTION F_VN_GetImageChannel : HRESULT
	VAR_INPUT
		ipSrcImage	:	ITcVnImage;	(* Source image *)
		ipDestImage	:	REFERENCE TO ITcVnImage;	(* Destination image (An appropriate image will be created if required.) *)
		nChannelIndex	:	UINT;	(* Index of the requested source image channel *)
		hrPrev	:	HRESULT;	(* HRESULT indicating the result of previous operations (If SUCCEEDED(hrPrev) equals false, no operation is executed.) *)
	END_VAR

END_FUNCTION

// Functions/Basic Image Operations/F_VN_GetImageHeight

	{attribute 'TcIecLibraryType'}
	{attribute 'external_name' := 'F_VN_GetImageHeight_GUID_0DEB5609_56D4_B77E_634C_3E0644346F9D'}
	(* Return the height of an image. (Alternatively use interface method .GetHeight.) *)
	FUNCTION F_VN_GetImageHeight : HRESULT
	VAR_INPUT
		ipImage	:	ITcVnImage;	(* Image *)
	END_VAR
	VAR_IN_OUT
		nHeight	:	UDINT;	(* Return the height of ipImage *)
	END_VAR
	VAR_INPUT
		hrPrev	:	HRESULT;	(* HRESULT indicating the result of previous operations (If SUCCEEDED(hrPrev) equals false, no operation is executed.) *)
	END_VAR

END_FUNCTION

// Functions/Basic Image Operations/F_VN_GetImageInfo

	{attribute 'TcIecLibraryType'}
	{attribute 'external_name' := 'F_VN_GetImageInfo_GUID_4CA6D81F_12B0_B0F2_72A2_044FF24AB2EE'}
	(* Gets a struct containing all common meta infos of the image. (Alternatively use interface method .GetImageInfo.) *)
	FUNCTION F_VN_GetImageInfo : HRESULT
	VAR_INPUT
		ipImage	:	ITcVnImage;	(* Image *)
	END_VAR
	VAR_IN_OUT
		stImageInfo	:	TcVnImageInfo;	(* Returns a struct describing the image *)
	END_VAR
	VAR_INPUT
		hrPrev	:	HRESULT;	(* HRESULT indicating the result of previous operations (If SUCCEEDED(hrPrev) equals false, no operation is executed.) *)
	END_VAR

END_FUNCTION

// Functions/Basic Image Operations/F_VN_GetImageWidth

	{attribute 'TcIecLibraryType'}
	{attribute 'external_name' := 'F_VN_GetImageWidth_GUID_3509AA6E_63E6_BB78_7F98_A569C4A4F477'}
	(* Return the width of an image. (Alternatively use interface method .GetWidth.) *)
	FUNCTION F_VN_GetImageWidth : HRESULT
	VAR_INPUT
		ipImage	:	ITcVnImage;	(* Image *)
	END_VAR
	VAR_IN_OUT
		nWidth	:	UDINT;	(* Return the width of ipImage *)
	END_VAR
	VAR_INPUT
		hrPrev	:	HRESULT;	(* HRESULT indicating the result of previous operations (If SUCCEEDED(hrPrev) equals false, no operation is executed.) *)
	END_VAR

END_FUNCTION

// Functions/Basic Image Operations/F_VN_GetPixel

	{attribute 'TcIecLibraryType'}
	{attribute 'external_name' := 'F_VN_GetPixel_GUID_37E0A656_6DB7_B118_68C1_1E84E3ACE452'}
	(* Gets a specific pixel. *)
	FUNCTION F_VN_GetPixel : HRESULT
	VAR_INPUT
		ipSrcImage	:	ITcVnImage;	(* Source image *)
	END_VAR
	VAR_IN_OUT
		aValue	:	TcVnVector4_LREAL;	(* Returns the pixel value (Unused channels are set to 0.) *)
	END_VAR
	VAR_INPUT
		nX	:	UDINT;	(* x coordinate of the pixel *)
		nY	:	UDINT;	(* y coordinate of the pixel *)
		hrPrev	:	HRESULT;	(* HRESULT indicating the result of previous operations (If SUCCEEDED(hrPrev) equals false, no operation is executed.) *)
	END_VAR

END_FUNCTION

// Functions/Basic Image Operations/F_VN_GetPixelFormat

	{attribute 'TcIecLibraryType'}
	{attribute 'external_name' := 'F_VN_GetPixelFormat_GUID_BCE8A3A0_41C2_B6F0_50C9_F48D3EE1C2D1'}
	(* Gets the pixel format of an image. (Alternatively use interface method .GetPixelFormat.) *)
	FUNCTION F_VN_GetPixelFormat : HRESULT
	VAR_INPUT
		ipImage	:	ITcVnImage;	(* Image *)
	END_VAR
	VAR_IN_OUT
		stPixelFormat	:	TcVnPixelFormat;	(* Returns a struct describing the pixel format *)
	END_VAR
	VAR_INPUT
		hrPrev	:	HRESULT;	(* HRESULT indicating the result of previous operations (If SUCCEEDED(hrPrev) equals false, no operation is executed.) *)
	END_VAR

END_FUNCTION

// Functions/Basic Image Operations/F_VN_GetRoi

	{attribute 'TcIecLibraryType'}
	{attribute 'external_name' := 'F_VN_GetRoi_GUID_7F4C3605_EB57_B2F7_6BB3_7CDC3AFB1F9B'}
	(* Gets the coordinates of the region of interest (ROI) within the image. *)
	FUNCTION F_VN_GetRoi : HRESULT
	VAR_INPUT
		ipSrcImage	:	ITcVnImage;	(* Source image *)
	END_VAR
	VAR_IN_OUT
		stRoi	:	TcVnRectangle_UDINT;	(* Returns the coordinates of the region of interest *)
	END_VAR
	VAR_INPUT
		hrPrev	:	HRESULT;	(* HRESULT indicating the result of previous operations (If SUCCEEDED(hrPrev) equals false, no operation is executed.) *)
	END_VAR

END_FUNCTION

// Functions/Basic Image Operations/F_VN_MixImageChannels

	{attribute 'TcIecLibraryType'}
	{attribute 'external_name' := 'F_VN_MixImageChannels_GUID_79CC9181_D4AA_B8E7_49AC_F10F1B350DA9'}
	(* Mix image channels by copying the specified channels of the source image into the specified channels of the destination image. *)
	FUNCTION F_VN_MixImageChannels : HRESULT
	VAR_INPUT
		ipSrcImage	:	ITcVnImage;	(* Source image *)
		ipDestImage	:	REFERENCE TO ITcVnImage;	(* Destination image (An appropriate image will be created if required.) *)
		ipIndicesFromTo	:	ITcVnContainer;	(* Index pairs (ContainerType_Vector_TcVnVector2_DINT), specifying which source channel (TcVnVector2_DINT [0]) should be copied to which destination channel (TcVnVector2_DINT [1]). *)
		hrPrev	:	HRESULT;	(* HRESULT indicating the result of previous operations (If SUCCEEDED(hrPrev) equals false, no operation is executed.) *)
	END_VAR

END_FUNCTION

// Functions/Basic Image Operations/F_VN_ResetRoi

	{attribute 'TcIecLibraryType'}
	{attribute 'external_name' := 'F_VN_ResetRoi_GUID_AFDC0572_CC81_BC24_7643_30D4B3D2F298'}
	(* Reset the region of interest (ROI) of an image. (After this operation, the ROI is set to the entire image.) *)
	FUNCTION F_VN_ResetRoi : HRESULT
	VAR_INPUT
		ipImage	:	ITcVnImage;	(* Image *)
		hrPrev	:	HRESULT;	(* HRESULT indicating the result of previous operations (If SUCCEEDED(hrPrev) equals false, no operation is executed.) *)
	END_VAR

END_FUNCTION

// Functions/Basic Image Operations/F_VN_SetImageChannel

	{attribute 'TcIecLibraryType'}
	{attribute 'external_name' := 'F_VN_SetImageChannel_GUID_899D2C8B_910A_B504_5E32_099D1FAB329D'}
	(* Sets the specified destination image channel to the values of the specified source image channel. *)
	FUNCTION F_VN_SetImageChannel : HRESULT
	VAR_INPUT
		ipSrcImage	:	ITcVnImage;	(* Source image *)
		ipDestImage	:	REFERENCE TO ITcVnImage;	(* Destination image (An appropriate image will be created if required.) *)
		nSrcChannelIndex	:	UINT;	(* Index of the source image channel *)
		nDestChannelIndex	:	UINT;	(* Index of the destination image channel, which will be replaced by the specified source image channel *)
		hrPrev	:	HRESULT;	(* HRESULT indicating the result of previous operations (If SUCCEEDED(hrPrev) equals false, no operation is executed.) *)
	END_VAR

END_FUNCTION

// Functions/Basic Image Operations/F_VN_SetPixel

	{attribute 'TcIecLibraryType'}
	{attribute 'external_name' := 'F_VN_SetPixel_GUID_08C80492_CB46_B15E_7934_A2DC47E02BAE'}
	(* Sets a specific pixel. *)
	FUNCTION F_VN_SetPixel : HRESULT
	VAR_INPUT
		ipSrcImage	:	ITcVnImage;	(* Source image *)
	END_VAR
	VAR_IN_OUT
		aValue	:	TcVnVector4_LREAL;	(* The pixel value to set (additional channels are ignored.) *)
	END_VAR
	VAR_INPUT
		nX	:	UDINT;	(* x coordinate of the pixel *)
		nY	:	UDINT;	(* y coordinate of the pixel *)
		hrPrev	:	HRESULT;	(* HRESULT indicating the result of previous operations (If SUCCEEDED(hrPrev) equals false, no operation is executed.) *)
	END_VAR

END_FUNCTION

// Functions/Basic Image Operations/F_VN_SetPixels

	{attribute 'TcIecLibraryType'}
	{attribute 'external_name' := 'F_VN_SetPixels_GUID_796F2676_AF97_BF9A_7FDF_B88266E30091'}
	(* Sets all pixels of an image to a given value. *)
	FUNCTION F_VN_SetPixels : HRESULT
	VAR_INPUT
		ipDestImage	:	ITcVnImage;	(* Destination image *)
	END_VAR
	VAR_IN_OUT
		aValue	:	TcVnVector4_LREAL;	(* Pixel value *)
	END_VAR
	VAR_INPUT
		hrPrev	:	HRESULT;	(* HRESULT indicating the result of previous operations (If SUCCEEDED(hrPrev) equals false, no operation is executed.) *)
	END_VAR

END_FUNCTION

// Functions/Basic Image Operations/F_VN_SetPixelsExp

	{attribute 'TcIecLibraryType'}
	{attribute 'external_name' := 'F_VN_SetPixelsExp_GUID_C6473839_89BA_B336_6B46_4D9AA061A50B'}
	(* Sets all pixels of an image to a given value. (expert function) *)
	FUNCTION F_VN_SetPixelsExp : HRESULT
	VAR_INPUT
		ipDestImage	:	ITcVnImage;	(* Destination image *)
	END_VAR
	VAR_IN_OUT
		aValue	:	TcVnVector4_LREAL;	(* Pixel value *)
	END_VAR
	VAR_INPUT
		ipMask	:	ITcVnImage;	(* Mask image *)
		hrPrev	:	HRESULT;	(* HRESULT indicating the result of previous operations (If SUCCEEDED(hrPrev) equals false, no operation is executed.) *)
	END_VAR

END_FUNCTION

// Functions/Basic Image Operations/F_VN_SetRoi

	{attribute 'TcIecLibraryType'}
	{attribute 'external_name' := 'F_VN_SetRoi_GUID_E8D3927C_1968_B545_63DB_8B4797F958AB'}
	(* Sets a region of interest (ROI) within an image. *)
	FUNCTION F_VN_SetRoi : HRESULT
	VAR_INPUT
		nX	:	UDINT;	(* Left boundary (inclusive 0-based index) *)
		nY	:	UDINT;	(* Upper boundary (inclusive 0-based index) *)
		nWidth	:	UDINT;	(* ROI width *)
		nHeight	:	UDINT;	(* ROI height *)
		ipDestImage	:	ITcVnImage;	(* Destination image *)
		hrPrev	:	HRESULT;	(* HRESULT indicating the result of previous operations (If SUCCEEDED(hrPrev) equals false, no operation is executed.) *)
	END_VAR

END_FUNCTION

// Functions/Basic Image Operations/F_VN_SetRoi_TcVnRectangle_DINT

	{attribute 'TcIecLibraryType'}
	{attribute 'external_name' := 'F_VN_SetRoi_TcVnRectangle_DINT_GUID_B698DF56_47D4_B38F_7A85_73AEAB072008'}
	(* Sets a region of interest (ROI) within an image. *)
	FUNCTION F_VN_SetRoi_TcVnRectangle_DINT : HRESULT
	VAR_IN_OUT
		stRoi	:	TcVnRectangle_DINT;	(* Region of interest *)
	END_VAR
	VAR_INPUT
		ipDestImage	:	ITcVnImage;	(* Destination image *)
		hrPrev	:	HRESULT;	(* HRESULT indicating the result of previous operations (If SUCCEEDED(hrPrev) equals false, no operation is executed.) *)
	END_VAR

END_FUNCTION

// Functions/Basic Image Operations/F_VN_SetRoi_TcVnRectangle_UDINT

	{attribute 'TcIecLibraryType'}
	{attribute 'external_name' := 'F_VN_SetRoi_TcVnRectangle_UDINT_GUID_E3A29C0E_EC80_B93E_7D26_A2ECE448239A'}
	(* Sets a region of interest (ROI) within an image. *)
	FUNCTION F_VN_SetRoi_TcVnRectangle_UDINT : HRESULT
	VAR_IN_OUT
		stRoi	:	TcVnRectangle_UDINT;	(* Region of interest *)
	END_VAR
	VAR_INPUT
		ipDestImage	:	ITcVnImage;	(* Destination image *)
		hrPrev	:	HRESULT;	(* HRESULT indicating the result of previous operations (If SUCCEEDED(hrPrev) equals false, no operation is executed.) *)
	END_VAR

END_FUNCTION

// Functions/Basic Image Operations/F_VN_SplitImageChannels

	{attribute 'TcIecLibraryType'}
	{attribute 'external_name' := 'F_VN_SplitImageChannels_GUID_2AD2A707_3CF0_BAAB_6FB3_2C29D43AD962'}
	(* Split a multi-channel image into multiple single channel images (1 for each source image channel). *)
	FUNCTION F_VN_SplitImageChannels : HRESULT
	VAR_INPUT
		ipSrcImage	:	ITcVnImage;	(* Source image with multiple channels *)
		pDestImages	:	PVOID;	(* Pointer to an array of ITcVnImage (appropriate destination images will be created if required) *)
		nArraySize	:	UINT;	(* Number of pDestImages array elements (array must be >= ipSourceImage channels) *)
		hrPrev	:	HRESULT;	(* HRESULT indicating the result of previous operations (If SUCCEEDED(hrPrev) equals false, no operation is executed.) *)
	END_VAR
	VAR_OUTPUT
		nImageChannels	:	UINT;	(* Actual source image channels *)
	END_VAR

END_FUNCTION

// Functions/Basic Image Operations/F_VN_TransformIntoDisplayableImageExp

	{attribute 'TcIecLibraryType'}
	{attribute 'external_name' := 'F_VN_TransformIntoDisplayableImageExp_GUID_95F6652F_D0D1_B1C2_6587_9DC3A044A515'}
	(* Transform an image into a displayable image. The source image will be released and zeroed while existing destination images will be released and overwritten with the function result. If bAllowDeepCopy equals false, the source image must not be used anywhere else and the transformation is always very fast. Otherwise, if bAllowDeepCopy equals true, a deep copy of the source image might be created if required, which will result in a longer execution time. If you want to use ipSrcImage after this function call, use F_VN_CopyIntoDisplayableImage instead. (expert function) *)
	FUNCTION F_VN_TransformIntoDisplayableImageExp : HRESULT
	VAR_INPUT
		ipSrcImage	:	REFERENCE TO ITcVnImage;	(* Source image *)
		ipDestImage	:	REFERENCE TO ITcVnDisplayableImage;	(* Returns the displayable image *)
		bAllowDeepCopy	:	BOOL;	(* Allow deep image copies, if required *)
		hrPrev	:	HRESULT;	(* HRESULT indicating the result of previous operations (If SUCCEEDED(hrPrev) equals false, no operation is executed.) *)
	END_VAR

END_FUNCTION

// Functions/Container Statistics/F_VN_ContainerAverage

	{attribute 'TcIecLibraryType'}
	{attribute 'external_name' := 'F_VN_ContainerAverage_GUID_2904C789_5402_B1C9_4EC0_C848213BD188'}
	(* Calculate the average of elements in a container. *)
	FUNCTION F_VN_ContainerAverage : HRESULT
	VAR_INPUT
		ipSrcContainer	:	ITcVnContainer;	(* Source container (Arithmetic, point and vector element types are supported. For points and vectors, the euclidean norm is used.) *)
	END_VAR
	VAR_IN_OUT
		fAverage	:	LREAL;	(* Returns the calculated average value *)
	END_VAR
	VAR_INPUT
		hrPrev	:	HRESULT;	(* HRESULT indicating the result of previous operations (If SUCCEEDED(hrPrev) equals false, no operation is executed.) *)
	END_VAR

END_FUNCTION

// Functions/Container Statistics/F_VN_ContainerAverageElementwise2

	{attribute 'TcIecLibraryType'}
	{attribute 'external_name' := 'F_VN_ContainerAverageElementwise2_GUID_261A77D6_849B_B33E_477A_4C7E294079CA'}
	(* Calculate the elementwise average of 2D elements in a container. *)
	FUNCTION F_VN_ContainerAverageElementwise2 : HRESULT
	VAR_INPUT
		ipSrcContainer	:	ITcVnContainer;	(* Source container with 2D points or vectors *)
	END_VAR
	VAR_IN_OUT
		aAverage	:	TcVnVector2_LREAL;	(* Returns the calculated average values *)
	END_VAR
	VAR_INPUT
		hrPrev	:	HRESULT;	(* HRESULT indicating the result of previous operations (If SUCCEEDED(hrPrev) equals false, no operation is executed.) *)
	END_VAR

END_FUNCTION

// Functions/Container Statistics/F_VN_ContainerAverageElementwise3

	{attribute 'TcIecLibraryType'}
	{attribute 'external_name' := 'F_VN_ContainerAverageElementwise3_GUID_C372ACF8_89E2_B96F_6253_1D85BDD8FDA8'}
	(* Calculate the elementwise average of 3D elements in a container. *)
	FUNCTION F_VN_ContainerAverageElementwise3 : HRESULT
	VAR_INPUT
		ipSrcContainer	:	ITcVnContainer;	(* Source container with 3D points or vectors *)
	END_VAR
	VAR_IN_OUT
		aAverage	:	TcVnVector3_LREAL;	(* Returns the calculated average values *)
	END_VAR
	VAR_INPUT
		hrPrev	:	HRESULT;	(* HRESULT indicating the result of previous operations (If SUCCEEDED(hrPrev) equals false, no operation is executed.) *)
	END_VAR

END_FUNCTION

// Functions/Container Statistics/F_VN_ContainerAverageElementwise4

	{attribute 'TcIecLibraryType'}
	{attribute 'external_name' := 'F_VN_ContainerAverageElementwise4_GUID_5D2003C2_3B53_B09B_4BCE_B4240FEE8CCA'}
	(* Calculate the elementwise average of 4D elements in a container. *)
	FUNCTION F_VN_ContainerAverageElementwise4 : HRESULT
	VAR_INPUT
		ipSrcContainer	:	ITcVnContainer;	(* Source container with 4D vectors *)
	END_VAR
	VAR_IN_OUT
		aAverage	:	TcVnVector4_LREAL;	(* Returns the calculated average values *)
	END_VAR
	VAR_INPUT
		hrPrev	:	HRESULT;	(* HRESULT indicating the result of previous operations (If SUCCEEDED(hrPrev) equals false, no operation is executed.) *)
	END_VAR

END_FUNCTION

// Functions/Container Statistics/F_VN_ContainerAverageVariance

	{attribute 'TcIecLibraryType'}
	{attribute 'external_name' := 'F_VN_ContainerAverageVariance_GUID_7BE1ABC3_C498_BDB7_4034_69FA1C0CAF28'}
	(* Calculate the average and variance of elements in a container. *)
	FUNCTION F_VN_ContainerAverageVariance : HRESULT
	VAR_INPUT
		ipSrcContainer	:	ITcVnContainer;	(* Source container (Arithmetic, point and vector element types are supported. For points and vectors, the euclidean norm is used.) *)
	END_VAR
	VAR_IN_OUT
		fAverage	:	LREAL;	(* Returns the calculated average value *)
		fVariance	:	LREAL;	(* Returns the calculated variance value *)
	END_VAR
	VAR_INPUT
		hrPrev	:	HRESULT;	(* HRESULT indicating the result of previous operations (If SUCCEEDED(hrPrev) equals false, no operation is executed.) *)
	END_VAR

END_FUNCTION

// Functions/Container Statistics/F_VN_ContainerAverageVarianceElementwise2

	{attribute 'TcIecLibraryType'}
	{attribute 'external_name' := 'F_VN_ContainerAverageVarianceElementwise2_GUID_1E542988_1F76_B642_4D68_14ABC3FFA6F1'}
	(* Calculate the elementwise average and variance of 2D elements in a container. *)
	FUNCTION F_VN_ContainerAverageVarianceElementwise2 : HRESULT
	VAR_INPUT
		ipSrcContainer	:	ITcVnContainer;	(* Source container with 2D points or vectors *)
	END_VAR
	VAR_IN_OUT
		aAverage	:	TcVnVector2_LREAL;	(* Returns the calculated average values *)
		aVariance	:	TcVnVector2_LREAL;	(* Returns the calculated variance values *)
	END_VAR
	VAR_INPUT
		hrPrev	:	HRESULT;	(* HRESULT indicating the result of previous operations (If SUCCEEDED(hrPrev) equals false, no operation is executed.) *)
	END_VAR

END_FUNCTION

// Functions/Container Statistics/F_VN_ContainerAverageVarianceElementwise3

	{attribute 'TcIecLibraryType'}
	{attribute 'external_name' := 'F_VN_ContainerAverageVarianceElementwise3_GUID_790FA727_AF02_BEAF_58F4_D92D932F49CD'}
	(* Calculate the elementwise average and variance of 3D elements in a container. *)
	FUNCTION F_VN_ContainerAverageVarianceElementwise3 : HRESULT
	VAR_INPUT
		ipSrcContainer	:	ITcVnContainer;	(* Source container with 3D points or vectors *)
	END_VAR
	VAR_IN_OUT
		aAverage	:	TcVnVector3_LREAL;	(* Returns the calculated average values *)
		aVariance	:	TcVnVector3_LREAL;	(* Returns the calculated variance values *)
	END_VAR
	VAR_INPUT
		hrPrev	:	HRESULT;	(* HRESULT indicating the result of previous operations (If SUCCEEDED(hrPrev) equals false, no operation is executed.) *)
	END_VAR

END_FUNCTION

// Functions/Container Statistics/F_VN_ContainerAverageVarianceElementwise4

	{attribute 'TcIecLibraryType'}
	{attribute 'external_name' := 'F_VN_ContainerAverageVarianceElementwise4_GUID_8092E4BB_1D67_B076_714C_885CA68F5781'}
	(* Calculate the elementwise average and variance of 4D elements in a container. *)
	FUNCTION F_VN_ContainerAverageVarianceElementwise4 : HRESULT
	VAR_INPUT
		ipSrcContainer	:	ITcVnContainer;	(* Source container with 4D vectors *)
	END_VAR
	VAR_IN_OUT
		aAverage	:	TcVnVector4_LREAL;	(* Returns the calculated average values *)
		aVariance	:	TcVnVector4_LREAL;	(* Returns the calculated variance values *)
	END_VAR
	VAR_INPUT
		hrPrev	:	HRESULT;	(* HRESULT indicating the result of previous operations (If SUCCEEDED(hrPrev) equals false, no operation is executed.) *)
	END_VAR

END_FUNCTION

// Functions/Container Statistics/F_VN_MaxElement

	{attribute 'TcIecLibraryType'}
	{attribute 'external_name' := 'F_VN_MaxElement_GUID_10DF45E8_4698_BF54_6120_B55870E6289F'}
	(* Gets the maximum element of a container. *)
	FUNCTION F_VN_MaxElement : HRESULT
	VAR_INPUT
		ipSrcContainer	:	ITcVnContainer;	(* Source container (Arithmetic, point and vector element types are supported. For points and vectors, the euclidean norm is used.) *)
		ipDestIterator	:	REFERENCE TO ITcVnBidirectionalIterator;	(* Returns an iterator to the requested element *)
	END_VAR
	VAR_IN_OUT
		nIndex	:	ULINT;	(* Returns the position of the requested element within the container *)
	END_VAR
	VAR_INPUT
		hrPrev	:	HRESULT;	(* HRESULT indicating the result of previous operations (If SUCCEEDED(hrPrev) equals false, no operation is executed.) *)
	END_VAR

END_FUNCTION

// Functions/Container Statistics/F_VN_MedianElement

	{attribute 'TcIecLibraryType'}
	{attribute 'external_name' := 'F_VN_MedianElement_GUID_F0CAFA6B_52D9_B111_7A5D_15CDCAC50B96'}
	(* Gets the median element of a container. *)
	FUNCTION F_VN_MedianElement : HRESULT
	VAR_INPUT
		ipSrcContainer	:	ITcVnContainer;	(* Source container (Arithmetic, point and vector element types are supported. For points and vectors, the euclidean norm is used.) *)
		ipDestIterator	:	REFERENCE TO ITcVnBidirectionalIterator;	(* Returns an iterator to the requested element *)
	END_VAR
	VAR_IN_OUT
		nIndex	:	ULINT;	(* Returns the position of the requested element within the container *)
	END_VAR
	VAR_INPUT
		hrPrev	:	HRESULT;	(* HRESULT indicating the result of previous operations (If SUCCEEDED(hrPrev) equals false, no operation is executed.) *)
	END_VAR

END_FUNCTION

// Functions/Container Statistics/F_VN_MinElement

	{attribute 'TcIecLibraryType'}
	{attribute 'external_name' := 'F_VN_MinElement_GUID_16EF1888_42B5_BD64_4512_195C3AF43EB1'}
	(* Gets the minimum element of a container. *)
	FUNCTION F_VN_MinElement : HRESULT
	VAR_INPUT
		ipSrcContainer	:	ITcVnContainer;	(* Source container (Arithmetic, point and vector element types are supported. For points and vectors, the euclidean norm is used.) *)
		ipDestIterator	:	REFERENCE TO ITcVnBidirectionalIterator;	(* Returns an iterator to the requested element *)
	END_VAR
	VAR_IN_OUT
		nIndex	:	ULINT;	(* Returns the position of the requested element within the container *)
	END_VAR
	VAR_INPUT
		hrPrev	:	HRESULT;	(* HRESULT indicating the result of previous operations (If SUCCEEDED(hrPrev) equals false, no operation is executed.) *)
	END_VAR

END_FUNCTION

// Functions/Fourier Analysis/F_VN_CreateBandpassButterworthFilter

	{attribute 'TcIecLibraryType'}
	{attribute 'external_name' := 'F_VN_CreateBandpassButterworthFilter_GUID_27FD6778_FF89_BCC5_4731_39379224D919'}
	(* Creates a bandpass Butterworth filter, which can be applied to a frequency domain image by element-wise multiplication. *)
	FUNCTION F_VN_CreateBandpassButterworthFilter : HRESULT
	VAR_INPUT
		ipFilter	:	REFERENCE TO ITcVnImage;	(* Returns the created filter (1 channel of type REAL or LREAL, depending on bDoublePrecision. Non-zero interface pointers are reused.). *)
		nWidth	:	UDINT;	(* Filter width (even, >= 2, must match the width of the image it is applied to) *)
		nHeight	:	UDINT;	(* Filter height (even, >= 2, must match the height of the image it is applied to) *)
		bDoublePrecision	:	BOOL;	(* If true, the filter is generated with double precision (LREAL) instead of single precision (REAL). *)
		bOriginAtCenter	:	BOOL;	(* If true, the filter origin is shifted to the image center. *)
		fCutoffDistance	:	LREAL;	(* The cutoff distance of the Butterworth filter (> 0). *)
		fBandWidth	:	LREAL;	(* The band width of the Butterworth filter (> 0). *)
		nOrder	:	UDINT;	(* The order of the Butterworth filter (> 0). *)
		fScale	:	LREAL;	(* The scale factor of the Butterworth filter denominator term (> 0, e.g. 0.414 or 1.0). *)
		hrPrev	:	HRESULT;	(* HRESULT indicating the result of previous operations (If SUCCEEDED(hrPrev) equals false, no operation is executed.) *)
	END_VAR

END_FUNCTION

// Functions/Fourier Analysis/F_VN_CreateBandpassGaussianFilter

	{attribute 'TcIecLibraryType'}
	{attribute 'external_name' := 'F_VN_CreateBandpassGaussianFilter_GUID_28B2F3B5_CD7A_BFBB_75E3_2F5E4C761EE6'}
	(* Creates a bandpass Gaussian filter, which can be applied to a frequency domain image by element-wise multiplication. *)
	FUNCTION F_VN_CreateBandpassGaussianFilter : HRESULT
	VAR_INPUT
		ipFilter	:	REFERENCE TO ITcVnImage;	(* Returns the created filter (1 channel of type REAL or LREAL, depending on bDoublePrecision. Non-zero interface pointers are reused.). *)
		nWidth	:	UDINT;	(* Filter width (even, >= 2, must match the width of the image it is applied to) *)
		nHeight	:	UDINT;	(* Filter height (even, >= 2, must match the height of the image it is applied to) *)
		bDoublePrecision	:	BOOL;	(* If true, the filter is generated with double precision (LREAL) instead of single precision (REAL). *)
		bOriginAtCenter	:	BOOL;	(* If true, the filter origin is shifted to the image center. *)
		fCutoffDistance	:	LREAL;	(* The cutoff distance of the Gaussian filter (> 0). *)
		fBandWidth	:	LREAL;	(* The band width of the Gaussian filter (> 0). *)
		hrPrev	:	HRESULT;	(* HRESULT indicating the result of previous operations (If SUCCEEDED(hrPrev) equals false, no operation is executed.) *)
	END_VAR

END_FUNCTION

// Functions/Fourier Analysis/F_VN_CreateBandrejectButterworthFilter

	{attribute 'TcIecLibraryType'}
	{attribute 'external_name' := 'F_VN_CreateBandrejectButterworthFilter_GUID_C071F030_55F2_BD22_6BF9_A439286AE858'}
	(* Creates a bandreject Butterworth filter, which can be applied to a frequency domain image by element-wise multiplication. *)
	FUNCTION F_VN_CreateBandrejectButterworthFilter : HRESULT
	VAR_INPUT
		ipFilter	:	REFERENCE TO ITcVnImage;	(* Returns the created filter (1 channel of type REAL or LREAL, depending on bDoublePrecision. Non-zero interface pointers are reused.). *)
		nWidth	:	UDINT;	(* Filter width (even, >= 2, must match the width of the image it is applied to) *)
		nHeight	:	UDINT;	(* Filter height (even, >= 2, must match the height of the image it is applied to) *)
		bDoublePrecision	:	BOOL;	(* If true, the filter is generated with double precision (LREAL) instead of single precision (REAL). *)
		bOriginAtCenter	:	BOOL;	(* If true, the filter origin is shifted to the image center. *)
		fCutoffDistance	:	LREAL;	(* The cutoff distance of the Butterworth filter (> 0). *)
		fBandWidth	:	LREAL;	(* The band width of the Butterworth filter (> 0). *)
		nOrder	:	UDINT;	(* The order of the Butterworth filter (> 0). *)
		fScale	:	LREAL;	(* The scale factor of the Butterworth filter denominator term (> 0, e.g. 0.414 or 1.0). *)
		hrPrev	:	HRESULT;	(* HRESULT indicating the result of previous operations (If SUCCEEDED(hrPrev) equals false, no operation is executed.) *)
	END_VAR

END_FUNCTION

// Functions/Fourier Analysis/F_VN_CreateBandrejectGaussianFilter

	{attribute 'TcIecLibraryType'}
	{attribute 'external_name' := 'F_VN_CreateBandrejectGaussianFilter_GUID_AE8FF277_AB4F_BF12_7B9B_E1BC80448E9B'}
	(* Creates a bandreject Gaussian filter, which can be applied to a frequency domain image by element-wise multiplication. *)
	FUNCTION F_VN_CreateBandrejectGaussianFilter : HRESULT
	VAR_INPUT
		ipFilter	:	REFERENCE TO ITcVnImage;	(* Returns the created filter (1 channel of type REAL or LREAL, depending on bDoublePrecision. Non-zero interface pointers are reused.). *)
		nWidth	:	UDINT;	(* Filter width (even, >= 2, must match the width of the image it is applied to) *)
		nHeight	:	UDINT;	(* Filter height (even, >= 2, must match the height of the image it is applied to) *)
		bDoublePrecision	:	BOOL;	(* If true, the filter is generated with double precision (LREAL) instead of single precision (REAL). *)
		bOriginAtCenter	:	BOOL;	(* If true, the filter origin is shifted to the image center. *)
		fCutoffDistance	:	LREAL;	(* The cutoff distance of the Gaussian filter (> 0). *)
		fBandWidth	:	LREAL;	(* The band width of the Gaussian filter (> 0). *)
		hrPrev	:	HRESULT;	(* HRESULT indicating the result of previous operations (If SUCCEEDED(hrPrev) equals false, no operation is executed.) *)
	END_VAR

END_FUNCTION

// Functions/Fourier Analysis/F_VN_CreateHighpassButterworthFilter

	{attribute 'TcIecLibraryType'}
	{attribute 'external_name' := 'F_VN_CreateHighpassButterworthFilter_GUID_A5BDA64D_ABF6_B146_6C07_49E2DCE7BDF0'}
	(* Creates a highpass Butterworth filter, which can be applied to a frequency domain image by element-wise multiplication. *)
	FUNCTION F_VN_CreateHighpassButterworthFilter : HRESULT
	VAR_INPUT
		ipFilter	:	REFERENCE TO ITcVnImage;	(* Returns the created filter (1 channel of type REAL or LREAL, depending on bDoublePrecision. Non-zero interface pointers are reused.). *)
		nWidth	:	UDINT;	(* Filter width (even, >= 2, must match the width of the image it is applied to) *)
		nHeight	:	UDINT;	(* Filter height (even, >= 2, must match the height of the image it is applied to) *)
		bDoublePrecision	:	BOOL;	(* If true, the filter is generated with double precision (LREAL) instead of single precision (REAL). *)
		bOriginAtCenter	:	BOOL;	(* If true, the filter origin is shifted to the image center. *)
		fCutoffDistance	:	LREAL;	(* The cutoff distance of the Butterworth filter (> 0). *)
		nOrder	:	UDINT;	(* The order of the Butterworth filter (> 0). *)
		fScale	:	LREAL;	(* The scale factor of the Butterworth filter denominator term (> 0, e.g. 0.414 or 1.0). *)
		hrPrev	:	HRESULT;	(* HRESULT indicating the result of previous operations (If SUCCEEDED(hrPrev) equals false, no operation is executed.) *)
	END_VAR

END_FUNCTION

// Functions/Fourier Analysis/F_VN_CreateHighpassGaussianFilter

	{attribute 'TcIecLibraryType'}
	{attribute 'external_name' := 'F_VN_CreateHighpassGaussianFilter_GUID_1239386C_21D5_BD4B_4D57_6DDBA6C52C01'}
	(* Creates a highpass Gaussian filter, which can be applied to a frequency domain image by element-wise multiplication. *)
	FUNCTION F_VN_CreateHighpassGaussianFilter : HRESULT
	VAR_INPUT
		ipFilter	:	REFERENCE TO ITcVnImage;	(* Returns the created filter (1 channel of type REAL or LREAL, depending on bDoublePrecision. Non-zero interface pointers are reused.). *)
		nWidth	:	UDINT;	(* Filter width (even, >= 2, must match the width of the image it is applied to) *)
		nHeight	:	UDINT;	(* Filter height (even, >= 2, must match the height of the image it is applied to) *)
		bDoublePrecision	:	BOOL;	(* If true, the filter is generated with double precision (LREAL) instead of single precision (REAL). *)
		bOriginAtCenter	:	BOOL;	(* If true, the filter origin is shifted to the image center. *)
		fCutoffDistance	:	LREAL;	(* The cutoff distance of the Gaussian filter (> 0). *)
		hrPrev	:	HRESULT;	(* HRESULT indicating the result of previous operations (If SUCCEEDED(hrPrev) equals false, no operation is executed.) *)
	END_VAR

END_FUNCTION

// Functions/Fourier Analysis/F_VN_CreateLowpassButterworthFilter

	{attribute 'TcIecLibraryType'}
	{attribute 'external_name' := 'F_VN_CreateLowpassButterworthFilter_GUID_B4BC6B04_F1D6_BA3D_607D_96E699A396DE'}
	(* Creates a lowpass Butterworth filter, which can be applied to a frequency domain image by element-wise multiplication. *)
	FUNCTION F_VN_CreateLowpassButterworthFilter : HRESULT
	VAR_INPUT
		ipFilter	:	REFERENCE TO ITcVnImage;	(* Returns the created filter (1 channel of type REAL or LREAL, depending on bDoublePrecision. Non-zero interface pointers are reused.). *)
		nWidth	:	UDINT;	(* Filter width (even, >= 2, must match the width of the image it is applied to) *)
		nHeight	:	UDINT;	(* Filter height (even, >= 2, must match the height of the image it is applied to) *)
		bDoublePrecision	:	BOOL;	(* If true, the filter is generated with double precision (LREAL) instead of single precision (REAL). *)
		bOriginAtCenter	:	BOOL;	(* If true, the filter origin is shifted to the image center. *)
		fCutoffDistance	:	LREAL;	(* The cutoff distance of the Butterworth filter (> 0). *)
		nOrder	:	UDINT;	(* The order of the Butterworth filter (> 0). *)
		fScale	:	LREAL;	(* The scale factor of the Butterworth filter denominator term (> 0, e.g. 0.414 or 1.0). *)
		hrPrev	:	HRESULT;	(* HRESULT indicating the result of previous operations (If SUCCEEDED(hrPrev) equals false, no operation is executed.) *)
	END_VAR

END_FUNCTION

// Functions/Fourier Analysis/F_VN_CreateLowpassGaussianFilter

	{attribute 'TcIecLibraryType'}
	{attribute 'external_name' := 'F_VN_CreateLowpassGaussianFilter_GUID_7FBAA138_CF43_B406_4315_723AE0B284C0'}
	(* Creates a lowpass Gaussian filter, which can be applied to a frequency domain image by element-wise multiplication. *)
	FUNCTION F_VN_CreateLowpassGaussianFilter : HRESULT
	VAR_INPUT
		ipFilter	:	REFERENCE TO ITcVnImage;	(* Returns the created filter (1 channel of type REAL or LREAL, depending on bDoublePrecision. Non-zero interface pointers are reused.). *)
		nWidth	:	UDINT;	(* Filter width (even, >= 2, must match the width of the image it is applied to) *)
		nHeight	:	UDINT;	(* Filter height (even, >= 2, must match the height of the image it is applied to) *)
		bDoublePrecision	:	BOOL;	(* If true, the filter is generated with double precision (LREAL) instead of single precision (REAL). *)
		bOriginAtCenter	:	BOOL;	(* If true, the filter origin is shifted to the image center. *)
		fCutoffDistance	:	LREAL;	(* The cutoff distance of the Gaussian filter (> 0). *)
		hrPrev	:	HRESULT;	(* HRESULT indicating the result of previous operations (If SUCCEEDED(hrPrev) equals false, no operation is executed.) *)
	END_VAR

END_FUNCTION

// Functions/Fourier Analysis/F_VN_Dft

	{attribute 'TcIecLibraryType'}
	{attribute 'external_name' := 'F_VN_Dft_GUID_1F5E1E3A_4DD5_B63F_457F_DB52DC1E993F'}
	(* Computes the DFT for a given image. *)
	FUNCTION F_VN_Dft : HRESULT
	VAR_INPUT
		ipSpatialImage	:	ITcVnImage;	(* Source image (elements of type REAL or LREAL, 1 (Re) or 2 (Re + Im) channels) *)
		ipFrequencyImage	:	REFERENCE TO ITcVnImage;	(* Destination image (same type as ipSpatialImage, but number of channels and size can vary depending on bPackedCCS and bAutoPadding. *)
		bPackedCCS	:	BOOL;	(* If true and ipSpatialImage has only 1 channel, the result image will have 1 channel with packed complex-conjugate-symmetrical format results. Otherwise, the result image will have 2 separate channels (Re + Im), containing the full spectrum. *)
		bAutoPadding	:	BOOL;	(* If true, the input image is automatically padded (with 0s) to optimal size if required, to speed up dft (Creates a temporary copy so that ipSpatialImage content stays unchanged, which also requires some additional computation power. Therefore, it is recommended to compare execution times with and without padding.) *)
		hrPrev	:	HRESULT;	(* HRESULT indicating the result of previous operations (If SUCCEEDED(hrPrev) equals false, no operation is executed.) *)
	END_VAR

END_FUNCTION

// Functions/Fourier Analysis/F_VN_InverseDft

	{attribute 'TcIecLibraryType'}
	{attribute 'external_name' := 'F_VN_InverseDft_GUID_D21C3C02_F052_B784_6481_43C6728A2E8D'}
	(* Compute the inverse DFT for a given frequency image. *)
	FUNCTION F_VN_InverseDft : HRESULT
	VAR_INPUT
		ipFrequencyImage	:	ITcVnImage;	(* Source frequency image (elements of type REAL or LREAL, 1 (packed CCS) or 2 (Re + Im) channels) *)
		ipSpatialImage	:	REFERENCE TO ITcVnImage;	(* Destination image (Same type as ipFrequencyImage, but number of channels can vary depending on bRealOutput. An appropriate image will be created if required.) *)
		bRealOutput	:	BOOL;	(* Only relevant if ipFrequencyImage has 2 channels. If true, the result image will have only 1 channel. Otherwise, the result image will have 2 separate channels (Re + Im). If ipFrequencyImage has only 1 channel, packed CCS format is assumed and the result image will always have only 1 channel. *)
		hrPrev	:	HRESULT;	(* HRESULT indicating the result of previous operations (If SUCCEEDED(hrPrev) equals false, no operation is executed.) *)
	END_VAR

END_FUNCTION

// Functions/Fourier Analysis/F_VN_OptimalDftSize

	{attribute 'TcIecLibraryType'}
	{attribute 'external_name' := 'F_VN_OptimalDftSize_GUID_FCFE53EE_2CEF_B975_5E4B_88F3DF754C99'}
	(* Computes the optimal image size for applying a dft (can lead to better performance). *)
	FUNCTION F_VN_OptimalDftSize : HRESULT
	VAR_INPUT
		ipImage	:	ITcVnImage;	(* Source image for which to compute the optimal width and height *)
	END_VAR
	VAR_IN_OUT
		nOptWidth	:	UDINT;	(* Returns the optimal width of the image *)
		nOptHeight	:	UDINT;	(* Returns the optimal height of the image *)
	END_VAR
	VAR_INPUT
		hrPrev	:	HRESULT;	(* HRESULT indicating the result of previous operations (If SUCCEEDED(hrPrev) equals false, no operation is executed.) *)
	END_VAR

END_FUNCTION

// Functions/Fourier Analysis/F_VN_PadImageBorder

	{attribute 'TcIecLibraryType'}
	{attribute 'external_name' := 'F_VN_PadImageBorder_GUID_81439A37_D4A4_B4AF_62AA_2630A3DD3286'}
	(* Add padding (zeros) around the original image borders. *)
	FUNCTION F_VN_PadImageBorder : HRESULT
	VAR_INPUT
		ipSrcImage	:	ITcVnImage;	(* Source image *)
		ipPaddedImage	:	REFERENCE TO ITcVnImage;	(* Padded destination image (Same type as ipSrcImage, an appropriate destination image will be created if required.) *)
		nTopBorder	:	UDINT;	(* Padding height in pixels above top border *)
		nBottomBorder	:	UDINT;	(* Padding height in pixels below bottom border *)
		nLeftBorder	:	UDINT;	(* Padding width in pixels before left border *)
		nRightBorder	:	UDINT;	(* Padding width in pixels after right border *)
		hrPrev	:	HRESULT;	(* HRESULT indicating the result of previous operations (If SUCCEEDED(hrPrev) equals false, no operation is executed.) *)
	END_VAR

END_FUNCTION

// Functions/Fourier Analysis/F_VN_PadImageBorderExp

	{attribute 'TcIecLibraryType'}
	{attribute 'external_name' := 'F_VN_PadImageBorderExp_GUID_26692D80_E211_B188_6068_D5271B1F402B'}
	(* Add padding around the original image borders. (expert function) *)
	FUNCTION F_VN_PadImageBorderExp : HRESULT
	VAR_INPUT
		ipSrcImage	:	ITcVnImage;	(* Source image *)
		ipPaddedImage	:	REFERENCE TO ITcVnImage;	(* Padded destination image (Same type as ipSrcImage, an appropriate destination image will be created if required.) *)
		nTopBorder	:	UDINT;	(* Padding height in pixels above top border *)
		nBottomBorder	:	UDINT;	(* Padding height in pixels below bottom border *)
		nLeftBorder	:	UDINT;	(* Padding width in pixels before left border *)
		nRightBorder	:	UDINT;	(* Padding width in pixels after right border *)
		ePaddingType	:	ETcVnBorderInterpolationMethod;	(* Specifies how the pixel values of the padding area are determined *)
	END_VAR
	VAR_IN_OUT
		aPaddingValue	:	TcVnVector4_LREAL;	(* Specifies the padding value if CONSTANT is used *)
	END_VAR
	VAR_INPUT
		hrPrev	:	HRESULT;	(* HRESULT indicating the result of previous operations (If SUCCEEDED(hrPrev) equals false, no operation is executed.) *)
	END_VAR

END_FUNCTION

// Functions/Machine Learning/F_VN_CreateBoostClassifier

	{attribute 'TcIecLibraryType'}
	{attribute 'external_name' := 'F_VN_CreateBoostClassifier_GUID_5D199503_0944_BC76_6657_620450DCAEFA'}
	(* Create a Boost classifier using the default parameters. The initial reference count is set to one if a new model is created and kept, otherwise. The Boost classifier is only applicable to binary classification problems. It learns to distinguish between samples labelled with two user-defined class labels by incrementally adding weak classifiers to improve the classification results. Models of this type neither support on-line training (sample by sample) nor retraining. *)
	FUNCTION F_VN_CreateBoostClassifier : HRESULT
	VAR_INPUT
		ipMlModel	:	REFERENCE TO ITcVnMlModel;	(* Returns the created model (Non-zero interface pointers are reused.) *)
		hrPrev	:	HRESULT;	(* HRESULT indicating the result of previous operations (If SUCCEEDED(hrPrev) equals false, no operation is executed.) *)
	END_VAR

END_FUNCTION

// Functions/Machine Learning/F_VN_CreateBoostClassifierExp

	{attribute 'TcIecLibraryType'}
	{attribute 'external_name' := 'F_VN_CreateBoostClassifierExp_GUID_583C2BBD_E827_B4D3_73C5_A89917A2145A'}
	(* Create a Boost classifier. The initial reference count is set to one if a new model is created and kept, otherwise. The Boost classifier is only applicable to binary classification problems. It learns to distinguish between samples labelled with two user-defined class labels by incrementally adding weak classifiers to improve the classification results. Models of this type neither support on-line training (sample by sample) nor retraining. (expert function) *)
	FUNCTION F_VN_CreateBoostClassifierExp : HRESULT
	VAR_INPUT
		ipMlModel	:	REFERENCE TO ITcVnMlModel;	(* Returns the created model (Non-zero interface pointers are reused.) *)
		eType	:	ETcVnBoostClassifierType;	(* Learning algorithm type (default: TCVN_BCT_REAL) *)
		nMaxDepth	:	UDINT;	(* Maximum tree depth (default: 1) *)
		nMinSamples	:	UDINT;	(* Minimum number of samples within a node required for splitting (default: 10) *)
		nWeakClassifiers	:	UDINT;	(* Number of weak classifiers (default: 100) *)
		fWeightTrimRate	:	LREAL;	(* Weight threshold used during training (off: 0; default: 0.95). *)
		hrPrev	:	HRESULT;	(* HRESULT indicating the result of previous operations (If SUCCEEDED(hrPrev) equals false, no operation is executed.) *)
	END_VAR

END_FUNCTION

// Functions/Machine Learning/F_VN_CreateBoostClassifierExp2

	{attribute 'TcIecLibraryType'}
	{attribute 'external_name' := 'F_VN_CreateBoostClassifierExp2_GUID_EC23561C_036E_BBCE_6181_EBB283FF5585'}
	(* Create a Boost classifier. The initial reference count is set to one if a new model is created and kept, otherwise. The Boost classifier is only applicable to binary classification problems. It learns to distinguish between samples labelled with two user-defined class labels by incrementally adding weak classifiers to improve the classification results. Models of this type neither support on-line training (sample by sample) nor retraining. (expert function) *)
	FUNCTION F_VN_CreateBoostClassifierExp2 : HRESULT
	VAR_INPUT
		ipMlModel	:	REFERENCE TO ITcVnMlModel;	(* Returns the created model (Non-zero interface pointers are reused.) *)
		eType	:	ETcVnBoostClassifierType;	(* Learning algorithm type (default: TCVN_BCT_REAL) *)
		nMaxDepth	:	UDINT;	(* Maximum tree depth (default: 1) *)
		nMinSamples	:	UDINT;	(* Minimum number of samples within a node required for splitting (default: 10) *)
		nWeakClassifiers	:	UDINT;	(* Number of weak classifiers (default: 100) *)
		fWeightTrimRate	:	LREAL;	(* Weight threshold used during training (off: 0; default: 0.95). *)
		ipClassPriors	:	ITcVnContainer;	(* Class priors (ContainerType_Vector_REAL or ContainerType_Vector_LREAL; only for classifiers; optional, set to 0 if not required or not allowed; default: 0) *)
		hrPrev	:	HRESULT;	(* HRESULT indicating the result of previous operations (If SUCCEEDED(hrPrev) equals false, no operation is executed.) *)
	END_VAR

END_FUNCTION

// Functions/Machine Learning/F_VN_CreateKmppModel

	{attribute 'TcIecLibraryType'}
	{attribute 'external_name' := 'F_VN_CreateKmppModel_GUID_7FBD24FA_20C6_B3FB_5CD1_D7785962541F'}
	(* Create a k-means++ model of the specified type. The initial reference count is set to one if a new model is created and kept, otherwise. Models of this type neither support on-line training (sample by sample) nor retraining. *)
	FUNCTION F_VN_CreateKmppModel : HRESULT
	VAR_INPUT
		ipMlModel	:	REFERENCE TO ITcVnMlModel;	(* Returns the created model (Non-zero interface pointers are reused.) *)
		eKmppType	:	ETcVnPrototypeClusterer;	(* k-means++ model type *)
		nK	:	UDINT;	(* Parameter k (number of clusters) *)
		hrPrev	:	HRESULT;	(* HRESULT indicating the result of previous operations (If SUCCEEDED(hrPrev) equals false, no operation is executed.) *)
	END_VAR

END_FUNCTION

// Functions/Machine Learning/F_VN_CreateKmppModelExp

	{attribute 'TcIecLibraryType'}
	{attribute 'external_name' := 'F_VN_CreateKmppModelExp_GUID_12EBE6DC_C464_BCD8_77AA_434DC7839617'}
	(* Create a k-means++ model of the specified type. The initial reference count is set to one if a new model is created and kept, otherwise. Models of this type neither support on-line training (sample by sample) nor retraining. (expert function) *)
	FUNCTION F_VN_CreateKmppModelExp : HRESULT
	VAR_INPUT
		ipMlModel	:	REFERENCE TO ITcVnMlModel;	(* Returns the created model (Non-zero interface pointers are reused.) *)
		eKmppType	:	ETcVnPrototypeClusterer;	(* k-means++ model type *)
		nK	:	UDINT;	(* Parameter k (number of clusters) *)
		bDoublePrecision	:	BOOL;	(* If true, the model is generated with double precision (LREAL) instead of single precision (REAL). (default: FALSE) *)
		nMaxIterations	:	UDINT;	(* Maximum number of iterations (triggers the usage of the default value of 10 if it equals 0) *)
		fEpsilon	:	LREAL;	(* Maximum allowed difference of the error between two successive iterations (triggers the usage of the default value of 0.001 if it equals 0) *)
		hrPrev	:	HRESULT;	(* HRESULT indicating the result of previous operations (If SUCCEEDED(hrPrev) equals false, no operation is executed.) *)
	END_VAR

END_FUNCTION

// Functions/Machine Learning/F_VN_CreateKnnModel

	{attribute 'TcIecLibraryType'}
	{attribute 'external_name' := 'F_VN_CreateKnnModel_GUID_BC495A11_E799_BFC7_760F_EEC0DFF6A157'}
	(* Create a k-nearest neighbors model of the specified type. The initial reference count is set to one if a new model is created and kept, otherwise. Models of this type support on-line training (sample by sample) and retraining. Predictions can only be scalar. *)
	FUNCTION F_VN_CreateKnnModel : HRESULT
	VAR_INPUT
		ipMlModel	:	REFERENCE TO ITcVnMlModel;	(* Returns the created model (Non-zero interface pointers are reused.) *)
		eKnnType	:	ETcVnKnn;	(* k-nearest neighbors model type *)
		nK	:	UDINT;	(* Parameter k used for prediction (number of considered neighbors) *)
		hrPrev	:	HRESULT;	(* HRESULT indicating the result of previous operations (If SUCCEEDED(hrPrev) equals false, no operation is executed.) *)
	END_VAR

END_FUNCTION

// Functions/Machine Learning/F_VN_CreateLbgModel

	{attribute 'TcIecLibraryType'}
	{attribute 'external_name' := 'F_VN_CreateLbgModel_GUID_2B13EB9A_FD90_BD13_6D1D_7BF0941071EF'}
	(* Create a LBG model of the specified type. The initial reference count is set to one if a new model is created and kept, otherwise. Models of this type neither support on-line training (sample by sample) nor retraining. *)
	FUNCTION F_VN_CreateLbgModel : HRESULT
	VAR_INPUT
		ipMlModel	:	REFERENCE TO ITcVnMlModel;	(* Returns the created model (Non-zero interface pointers are reused.) *)
		eLbgType	:	ETcVnPrototypeClusterer;	(* LBG model type *)
		nMaxClusters	:	UDINT;	(* Maximum number of clusters *)
		fMaxClusterRadius	:	LREAL;	(* Maximum allowed radius (L2 norm) of a single cluster, i.e. clusters with a higher radius will be split into smaller ones, until a global number of nMaxClusters is reached. *)
		bSingleSplitSteps	:	BOOL;	(* If true, the global optimization is always run after a single cluster has been split. If false, several clusters are split within the same step before applying the global optimization. Applying the global optimization less often is faster, but can lead to less optimal results, especially having 2 nearby clusters that could be represented by 1. *)
		hrPrev	:	HRESULT;	(* HRESULT indicating the result of previous operations (If SUCCEEDED(hrPrev) equals false, no operation is executed.) *)
	END_VAR

END_FUNCTION

// Functions/Machine Learning/F_VN_CreateLbgModelExp

	{attribute 'TcIecLibraryType'}
	{attribute 'external_name' := 'F_VN_CreateLbgModelExp_GUID_FE0CCAEA_9013_BCD3_5150_74D5D1AB6CA9'}
	(* Create a LBG model of the specified type. The initial reference count is set to one if a new model is created and kept, otherwise. Models of this type neither support on-line training (sample by sample) nor retraining. (expert function) *)
	FUNCTION F_VN_CreateLbgModelExp : HRESULT
	VAR_INPUT
		ipMlModel	:	REFERENCE TO ITcVnMlModel;	(* Returns the created model (Non-zero interface pointers are reused.) *)
		eLbgType	:	ETcVnPrototypeClusterer;	(* LBG model type *)
		nMaxClusters	:	UDINT;	(* Maximum number of clusters *)
		fMaxClusterRadius	:	LREAL;	(* Maximum allowed radius (L2 norm) of a single cluster, i.e. clusters with a higher radius will be split into smaller ones, until a global number of nMaxClusters is reached. *)
		bSingleSplitSteps	:	BOOL;	(* If true, the global optimization is always run after a single cluster has been split. If false, several clusters are split within the same step before applying the global optimization. Applying the global optimization less often is faster, but can lead to less optimal results, especially having 2 nearby clusters that could be represented by 1. *)
		bDoublePrecision	:	BOOL;	(* If true, the model is generated with double precision (LREAL) instead of single precision (REAL). (default: FALSE) *)
		nMaxIterations	:	UDINT;	(* Maximum number of iterations (triggers the usage of the default value of 10 if it equals 0) *)
		fEpsilon	:	LREAL;	(* Maximum allowed difference of the error between two successive iterations (triggers the usage of the default value of 0.001 if it equals 0) *)
		hrPrev	:	HRESULT;	(* HRESULT indicating the result of previous operations (If SUCCEEDED(hrPrev) equals false, no operation is executed.) *)
	END_VAR

END_FUNCTION

// Functions/Machine Learning/F_VN_CreateLdaTransform

	{attribute 'TcIecLibraryType'}
	{attribute 'external_name' := 'F_VN_CreateLdaTransform_GUID_3C6296C2_E9AD_B4ED_6E2B_9E7503405703'}
	(* Create an LDA-based feature transform from the provided data. The number of samples must be >= the number of features and the number of classes must be >= 2. The initial reference count is set to one if a new model is created and kept, otherwise. *)
	FUNCTION F_VN_CreateLdaTransform : HRESULT
	VAR_INPUT
		ipMlModel	:	REFERENCE TO ITcVnMlModel;	(* Returns the created feature transform (Non-zero interface pointers are reused.) *)
		ipSamples	:	ITcUnknown;	(* Container holding a batch of input samples (ContainerType_Vector_Vector_REAL or ContainerType_Vector_Vector_LREAL) *)
		ipClasses	:	ITcVnContainer;	(* Class labels corresponding to the input samples (ContainerType_Vector_DINT) *)
		hrPrev	:	HRESULT;	(* HRESULT indicating the result of previous operations (If SUCCEEDED(hrPrev) equals false, no operation is executed.) *)
	END_VAR

END_FUNCTION

// Functions/Machine Learning/F_VN_CreateLdaTransformViaComponentNum

	{attribute 'TcIecLibraryType'}
	{attribute 'external_name' := 'F_VN_CreateLdaTransformViaComponentNum_GUID_1866BB21_E7CB_B9A3_7AC0_01403E09E5BE'}
	(* Create an LDA-based feature transform from the provided data where the number of components to be used is predefined. The number of samples must be >= the number of features and the number of classes must be >= 2. The initial reference count is set to one if a new model is created and kept, otherwise. (expert function) *)
	FUNCTION F_VN_CreateLdaTransformViaComponentNum : HRESULT
	VAR_INPUT
		ipMlModel	:	REFERENCE TO ITcVnMlModel;	(* Returns the created feature transform (Non-zero interface pointers are reused.) *)
		ipSamples	:	ITcUnknown;	(* Container holding a batch of input samples (ContainerType_Vector_Vector_REAL or ContainerType_Vector_Vector_LREAL) *)
		ipClasses	:	ITcVnContainer;	(* Class labels corresponding to the input samples (ContainerType_Vector_DINT) *)
		nComponentNum	:	UDINT;	(* Number of components (nComponentNum must be smaller than the number of classes. A value of 0 results in the automatic computation of the maximum number of components.) *)
		hrPrev	:	HRESULT;	(* HRESULT indicating the result of previous operations (If SUCCEEDED(hrPrev) equals false, no operation is executed.) *)
	END_VAR

END_FUNCTION

// Functions/Machine Learning/F_VN_CreateNbcModel

	{attribute 'TcIecLibraryType'}
	{attribute 'external_name' := 'F_VN_CreateNbcModel_GUID_598E3B7E_FBC3_BC69_7FAF_279D40022FFA'}
	(* Create a normal Bayes classifier of the specified type. The initial reference count is set to one if a new model is created and kept, otherwise. In order to train normal Bayes classifiers, a sufficiently high number of samples is required for each class. It depends on the number of features and the distribution of the data. Hence, it needs to be tested for each application. Models of this type do not support on-line training (sample by sample). For the retraining of such classifier models, the set of presented classes must be identical to the previous learning steps. Otherwise, an exception is raised. *)
	FUNCTION F_VN_CreateNbcModel : HRESULT
	VAR_INPUT
		ipMlModel	:	REFERENCE TO ITcVnMlModel;	(* Returns the created model (Non-zero interface pointers are reused.) *)
		eNbcType	:	ETcVnNbc;	(* Normal Bayes classifier type *)
		hrPrev	:	HRESULT;	(* HRESULT indicating the result of previous operations (If SUCCEEDED(hrPrev) equals false, no operation is executed.) *)
	END_VAR

END_FUNCTION

// Functions/Machine Learning/F_VN_CreatePcaTransform

	{attribute 'TcIecLibraryType'}
	{attribute 'external_name' := 'F_VN_CreatePcaTransform_GUID_59A8383E_3036_B344_49CB_AFC26CC59D3C'}
	(* Create a PCA-based feature transform from the provided data. The maximum number of principal components that can be computed equals the minimum of the number of samples and the number of features. The initial reference count is set to one if a new model is created and kept, otherwise. *)
	FUNCTION F_VN_CreatePcaTransform : HRESULT
	VAR_INPUT
		ipMlModel	:	REFERENCE TO ITcVnMlModel;	(* Returns the created feature transform (Non-zero interface pointers are reused.) *)
		ipSamples	:	ITcUnknown;	(* Container holding a batch of input samples (ContainerType_Vector_Vector_REAL or ContainerType_Vector_Vector_LREAL) *)
		hrPrev	:	HRESULT;	(* HRESULT indicating the result of previous operations (If SUCCEEDED(hrPrev) equals false, no operation is executed.) *)
	END_VAR

END_FUNCTION

// Functions/Machine Learning/F_VN_CreatePcaTransformViaComponentNum

	{attribute 'TcIecLibraryType'}
	{attribute 'external_name' := 'F_VN_CreatePcaTransformViaComponentNum_GUID_AB9CB397_9E1B_BC6D_5EAA_D6F99A689326'}
	(* Create a PCA-based feature transform from the provided data where the number of prinicpal components to be used is predefined. The maximum number of principal components that can be computed equals the minimum of the number of samples and the number of features. The initial reference count is set to one if a new model is created and kept, otherwise. (expert function) *)
	FUNCTION F_VN_CreatePcaTransformViaComponentNum : HRESULT
	VAR_INPUT
		ipMlModel	:	REFERENCE TO ITcVnMlModel;	(* Returns the created feature transform (Non-zero interface pointers are reused.) *)
		ipSamples	:	ITcUnknown;	(* Container holding a batch of input samples (ContainerType_Vector_Vector_REAL or ContainerType_Vector_Vector_LREAL) *)
		nComponentNum	:	UDINT;	(* Number of principal components (A value of 0 results in the automatic computation of the maximum number of components.) *)
		hrPrev	:	HRESULT;	(* HRESULT indicating the result of previous operations (If SUCCEEDED(hrPrev) equals false, no operation is executed.) *)
	END_VAR

END_FUNCTION

// Functions/Machine Learning/F_VN_CreatePcaTransformViaVariance

	{attribute 'TcIecLibraryType'}
	{attribute 'external_name' := 'F_VN_CreatePcaTransformViaVariance_GUID_9E8C4406_C07F_B8CA_7371_2EED241804C6'}
	(* Create a PCA-based feature transform from the provided data based on a given fraction of variance to be retained. The maximum number of principal components that can be computed equals the minimum of the number of samples and the number of features. The initial reference count is set to one if a new model is created and kept, otherwise. (expert function) *)
	FUNCTION F_VN_CreatePcaTransformViaVariance : HRESULT
	VAR_INPUT
		ipMlModel	:	REFERENCE TO ITcVnMlModel;	(* Returns the created feature transform (Non-zero interface pointers are reused.) *)
		ipSamples	:	ITcUnknown;	(* Container holding a batch of input samples (ContainerType_Vector_Vector_REAL or ContainerType_Vector_Vector_LREAL) *)
		fRetainedVariance	:	LREAL;	(* Fraction of variance that is to be retained by the PCA (A value of 1.0 signifies 100%.) *)
		hrPrev	:	HRESULT;	(* HRESULT indicating the result of previous operations (If SUCCEEDED(hrPrev) equals false, no operation is executed.) *)
	END_VAR

END_FUNCTION

// Functions/Machine Learning/F_VN_CreateRTreesModel

	{attribute 'TcIecLibraryType'}
	{attribute 'external_name' := 'F_VN_CreateRTreesModel_GUID_DD01E029_A3CB_B046_5379_AAE89BCB0437'}
	(* Create a random trees model of the specified type. The initial reference count is set to one if a new model is created and kept, otherwise. Models of this type neither support on-line training (sample by sample) nor retraining. Predictions can only be scalar. *)
	FUNCTION F_VN_CreateRTreesModel : HRESULT
	VAR_INPUT
		ipMlModel	:	REFERENCE TO ITcVnMlModel;	(* Returns the created model (Non-zero interface pointers are reused.) *)
		eRTreesType	:	ETcVnRTrees;	(* Random trees model type *)
		hrPrev	:	HRESULT;	(* HRESULT indicating the result of previous operations (If SUCCEEDED(hrPrev) equals false, no operation is executed.) *)
	END_VAR

END_FUNCTION

// Functions/Machine Learning/F_VN_CreateRTreesModelExp

	{attribute 'TcIecLibraryType'}
	{attribute 'external_name' := 'F_VN_CreateRTreesModelExp_GUID_37B5C282_963A_BC24_6778_9591C4448951'}
	(* Create a random trees model of the specified type. The initial reference count is set to one if a new model is created and kept, otherwise. Models of this type neither support on-line training (sample by sample) nor retraining. Predictions can only be scalar. (expert function) *)
	FUNCTION F_VN_CreateRTreesModelExp : HRESULT
	VAR_INPUT
		ipMlModel	:	REFERENCE TO ITcVnMlModel;	(* Returns the created model (Non-zero interface pointers are reused.) *)
		eRTreesType	:	ETcVnRTrees;	(* Random trees model type *)
		nMaxDepth	:	UDINT;	(* Maximum tree depth (default: 5) *)
		nMinSamples	:	UDINT;	(* Minimum number of samples within a node required for splitting (default: 10) *)
		nActiveVariables	:	UDINT;	(* Number of variables considered for splitting (0 means sqrt(total number of variables); default: 0) *)
		nMaxIterations	:	UDINT;	(* Maximum number of iterations (disabled if it equals 0 and fEpsilon is different from 0.0; triggers the usage of the default value of 50 if nMaxIterations and fEpsilon equal 0) *)
		fEpsilon	:	LREAL;	(* Maximum allowed difference of the error between two successive iterations (disabled if it equals 0.0 and nMaxIterations is different from 0; triggers the usage of the default value of 0.1 if nMaxIterations and fEpsilon equal 0) *)
		hrPrev	:	HRESULT;	(* HRESULT indicating the result of previous operations (If SUCCEEDED(hrPrev) equals false, no operation is executed.) *)
	END_VAR

END_FUNCTION

// Functions/Machine Learning/F_VN_CreateRTreesModelExp2

	{attribute 'TcIecLibraryType'}
	{attribute 'external_name' := 'F_VN_CreateRTreesModelExp2_GUID_48A6F8CE_D5A5_BDE6_7A93_97D64038B3ED'}
	(* Create a random trees model of the specified type. The initial reference count is set to one if a new model is created and kept, otherwise. Models of this type neither support on-line training (sample by sample) nor retraining. Predictions can only be scalar. (expert function) *)
	FUNCTION F_VN_CreateRTreesModelExp2 : HRESULT
	VAR_INPUT
		ipMlModel	:	REFERENCE TO ITcVnMlModel;	(* Returns the created model (Non-zero interface pointers are reused.) *)
		eRTreesType	:	ETcVnRTrees;	(* Random trees model type *)
		nMaxDepth	:	UDINT;	(* Maximum tree depth (default: 5) *)
		nMinSamples	:	UDINT;	(* Minimum number of samples within a node required for splitting (default: 10) *)
		nActiveVariables	:	UDINT;	(* Number of variables considered for splitting (0 means sqrt(total number of variables); default: 0) *)
		nMaxIterations	:	UDINT;	(* Maximum number of iterations (disabled if it equals 0 and fEpsilon is different from 0.0; triggers the usage of the default value of 50 if nMaxIterations and fEpsilon equal 0) *)
		fEpsilon	:	LREAL;	(* Maximum allowed difference of the error between two successive iterations (disabled if it equals 0.0 and nMaxIterations is different from 0; triggers the usage of the default value of 0.1 if nMaxIterations and fEpsilon equal 0) *)
		fRegressionAccuracy	:	REAL;	(* Termination criterion for regressors (only for regressors; set to default if not allowed; default: 0.0) *)
		ipClassPriors	:	ITcVnContainer;	(* Class priors (ContainerType_Vector_REAL or ContainerType_Vector_LREAL; only for classifiers; optional, set to 0 if not required or not allowed; default: 0) *)
		hrPrev	:	HRESULT;	(* HRESULT indicating the result of previous operations (If SUCCEEDED(hrPrev) equals false, no operation is executed.) *)
	END_VAR

END_FUNCTION

// Functions/Machine Learning/F_VN_CreateStaModel

